C03573=1020.006,186.866,-121.307,168.110,50.738,159.496
C03574=1020.013,187.146,-121.332,168.114,50.729,159.495
C03575=1020.018,187.428,-121.358,168.119,50.721,159.494
C03576=1020.024,187.709,-121.384,168.124,50.713,159.494
C03577=1020.030,187.990,-121.410,168.128,50.705,159.493
C03578=1020.035,188.240,-121.432,168.133,50.698,159.492
C03579=1020.040,188.488,-121.455,168.137,50.691,159.491
C03580=1020.045,188.738,-121.477,168.140,50.683,159.490
C03581=1020.050,188.986,-121.500,168.144,50.676,159.490
C03582=1020.056,189.235,-121.523,168.149,50.669,159.489
C03583=1020.061,189.484,-121.546,168.153,50.662,159.488
C03584=1020.066,189.733,-121.568,168.157,50.654,159.487
C03585=1020.071,189.982,-121.591,168.161,50.647,159.486
C03586=1020.076,190.230,-121.614,168.165,50.640,159.486
C03587=1020.081,190.480,-121.637,168.170,50.633,159.485
C03588=1020.087,190.729,-121.660,168.174,50.626,159.484
C03589=1020.092,190.977,-121.682,168.177,50.619,159.483
C03590=1020.097,191.226,-121.706,168.181,50.611,159.483
C03591=1020.102,191.475,-121.728,168.186,50.604,159.482
C03592=1020.108,191.724,-121.750,168.190,50.597,159.481
C03593=1020.113,191.973,-121.774,168.195,50.590,159.481
C03594=1020.118,192.222,-121.797,168.198,50.583,159.479
C03595=1020.123,192.470,-121.820,168.202,50.576,159.479
C03596=1020.128,192.720,-121.842,168.207,50.569,159.478
C03597=1020.134,192.969,-121.865,168.211,50.561,159.477
C03598=1020.139,193.217,-121.888,168.215,50.554,159.476
C03599=1020.144,193.466,-121.911,168.220,50.547,159.476
C03600=1020.150,193.715,-121.934,168.223,50.540,159.475
C03601=1020.155,193.964,-121.957,168.228,50.533,159.474
C03602=1020.160,194.213,-121.980,168.232,50.526,159.474
C03603=1020.165,194.462,-122.003,168.236,50.518,159.473
C03604=1020.171,194.711,-122.026,168.240,50.511,159.472
C03605=1020.175,194.959,-122.049,168.245,50.504,159.471
C03606=1020.181,195.208,-122.072,168.249,50.497,159.471
C03607=1020.187,195.457,-122.095,168.254,50.490,159.470
C03608=1020.192,195.706,-122.118,168.257,50.483,159.469
C03609=1020.198,195.955,-122.141,168.261,50.475,159.468
C03610=1020.203,196.203,-122.164,168.266,50.468,159.467
C03611=1020.208,196.453,-122.187,168.270,50.461,159.467
C03612=1020.213,196.702,-122.210,168.275,50.454,159.466
C03613=1020.219,196.950,-122.233,168.279,50.447,159.465
C03614=1020.224,197.200,-122.257,168.283,50.439,159.464
C03615=1020.229,197.448,-122.279,168.288,50.432,159.464
C03616=1020.235,197.697,-122.302,168.292,50.425,159.463
C03617=1020.240,197.946,-122.326,168.297,50.418,159.462
C03618=1020.246,198.195,-122.349,168.301,50.411,159.462
C03619=1020.251,198.444,-122.372,168.305,50.403,159.461
C03620=1020.256,198.693,-122.395,168.309,50.396,159.460
C03621=1020.262,198.941,-122.418,168.313,50.389,159.459
C03622=1020.267,199.190,-122.441,168.318,50.382,159.459
C03623=1020.272,199.439,-122.464,168.322,50.375,159.458
C03624=1020.277,199.688,-122.488,168.326,50.368,159.457
C03625=1020.283,199.937,-122.512,168.331,50.361,159.456
C03626=1020.288,200.186,-122.535,168.335,50.354,159.456
C03627=1020.293,200.435,-122.559,168.340,50.347,159.455
C03628=1020.299,200.684,-122.582,168.344,50.340,159.454
C03629=1020.304,200.932,-122.605,168.349,50.333,159.454
C03630=1020.309,201.181,-122.629,168.353,50.326,159.453
C03631=1020.314,201.430,-122.653,168.357,50.319,159.452
C03632=1020.320,201.679,-122.676,168.361,50.312,159.451
C03633=1020.325,201.928,-122.700,168.366,50.305,159.451
C03634=1020.330,202.176,-122.724,168.370,50.298,159.450
C03635=1020.336,202.425,-122.747,168.375,50.291,159.449
C03636=1020.341,202.674,-122.770,168.379,50.284,159.449
C03637=1020.346,202.923,-122.795,168.384,50.277,159.448
C03638=1020.368,203.963,-122.893,168.833,50.371,159.543
C03639=1020.373,204.181,-122.915,168.836,50.366,159.543
C03640=1020.379,204.400,-122.937,168.838,50.360,159.542
C03641=1020.384,204.618,-122.960,168.842,50.355,159.542
C03642=1020.390,204.838,-122.982,168.844,50.349,159.541
C03643=1020.396,205.057,-123.004,168.848,50.344,159.540
C03644=1020.401,205.276,-123.026,168.852,50.339,159.540
C03645=1020.406,205.494,-123.049,168.855,50.333,159.539
C03646=1020.412,205.713,-123.070,168.858,50.328,159.539
C03647=1020.418,205.961,-123.096,168.861,50.322,159.538
C03648=1020.424,206.210,-123.121,168.864,50.316,159.537
C03649=1020.431,206.459,-123.146,168.868,50.310,159.536
C03650=1020.437,206.707,-123.172,168.872,50.304,159.536
C03651=1020.443,206.956,-123.197,168.876,50.298,159.535
C03652=1020.449,207.204,-123.222,168.879,50.292,159.535
C03653=1020.455,207.453,-123.247,168.882,50.287,159.534
C03654=1020.461,207.701,-123.273,168.886,50.281,159.533
C03655=1020.466,207.950,-123.299,168.890,50.275,159.532
C03656=1020.473,208.198,-123.325,168.894,50.269,159.532
C03657=1020.479,208.447,-123.350,168.897,50.263,159.531
C03658=1020.485,208.696,-123.375,168.900,50.257,159.530
C03659=1020.492,208.944,-123.401,168.904,50.251,159.530
C03660=1020.498,209.193,-123.426,168.908,50.245,159.529
C03661=1020.504,209.442,-123.451,168.912,50.239,159.528
C03662=1020.510,209.690,-123.477,168.914,50.233,159.528
C03663=1020.516,209.939,-123.503,168.919,50.228,159.527
C03664=1020.522,210.187,-123.529,168.922,50.222,159.527
C03665=1020.528,210.436,-123.554,168.926,50.216,159.526
C03666=1020.535,210.685,-123.579,168.929,50.210,159.525
C03667=1020.540,210.933,-123.606,168.933,50.205,159.525
C03668=1020.547,211.182,-123.631,168.937,50.199,159.524
C03669=1020.553,211.431,-123.657,168.941,50.193,159.524
C03670=1020.559,211.680,-123.683,168.944,50.187,159.523
C03671=1020.565,211.928,-123.709,168.948,50.182,159.522
C03672=1020.572,212.177,-123.734,168.952,50.176,159.522
C03673=1020.577,212.426,-123.760,168.954,50.170,159.521
C03674=1020.584,212.674,-123.786,168.958,50.164,159.520
C03675=1020.590,212.923,-123.812,168.962,50.159,159.520
C03676=1020.596,213.171,-123.837,168.966,50.153,159.519
C03677=1020.602,213.420,-123.864,168.969,50.147,159.518
C03678=1020.608,213.668,-123.889,168.973,50.142,159.518
C03679=1020.614,213.916,-123.915,168.977,50.136,159.517
C03680=1020.620,214.165,-123.941,168.980,50.130,159.517
C03681=1020.626,214.414,-123.966,168.984,50.125,159.516
C03682=1020.633,214.663,-123.993,168.988,50.119,159.515
C03683=1020.639,214.912,-124.019,168.992,50.114,159.515
C03684=1020.645,215.160,-124.045,168.995,50.108,159.514
C03685=1020.651,215.408,-124.070,168.999,50.102,159.514
C03686=1020.657,215.657,-124.097,169.003,50.097,159.513
C03687=1020.663,215.905,-124.122,169.006,50.091,159.512
C03688=1020.670,216.154,-124.147,169.010,50.086,159.512
C03689=1020.676,216.403,-124.174,169.014,50.080,159.511
C03690=1020.682,216.652,-124.200,169.017,50.074,159.511
C03691=1020.689,216.900,-124.226,169.021,50.069,159.510
C03692=1020.694,217.149,-124.252,169.025,50.063,159.509
C03693=1020.701,217.397,-124.278,169.029,50.058,159.509
C03694=1020.707,217.646,-124.303,169.032,50.052,159.508
C03695=1020.714,217.894,-124.330,169.036,50.047,159.508
C03696=1020.720,218.143,-124.356,169.040,50.041,159.507
C03697=1020.726,218.391,-124.382,169.044,50.035,159.507
C03698=1020.732,218.640,-124.408,169.047,50.030,159.506
C03699=1020.737,218.861,-124.431,169.050,50.025,159.506
C03700=1020.743,219.082,-124.455,169.053,50.020,159.505
C03701=1020.748,219.304,-124.478,169.057,50.015,159.505
C03702=1020.754,219.525,-124.502,169.060,50.011,159.504
C03703=1020.759,219.747,-124.525,169.063,50.006,159.504
C03704=1020.764,219.968,-124.549,169.066,50.001,159.503
C03705=1020.770,220.190,-124.571,169.070,49.996,159.503
C03706=1020.775,220.410,-124.595,169.073,49.991,159.502
C03707=1020.781,220.659,-124.622,169.077,49.986,159.502
C03708=1020.788,220.908,-124.647,169.081,49.981,159.501
C03709=1020.794,221.157,-124.674,169.084,49.976,159.501
C03710=1020.800,221.405,-124.701,169.088,49.970,159.500
C03711=1020.806,221.653,-124.727,169.092,49.965,159.499
C03712=1020.812,221.902,-124.754,169.096,49.960,159.499
C03713=1020.819,222.151,-124.779,169.100,49.954,159.498
C03714=1020.824,222.399,-124.806,169.103,49.949,159.498
C03715=1020.830,222.647,-124.832,169.107,49.943,159.497
C03716=1020.837,222.896,-124.859,169.111,49.938,159.497
C03717=1020.843,223.144,-124.885,169.114,49.933,159.496
C03718=1020.849,223.393,-124.912,169.118,49.927,159.496
C03719=1020.856,223.642,-124.938,169.121,49.922,159.495
C03720=1020.861,223.891,-124.964,169.126,49.917,159.495
C03721=1020.868,224.139,-124.991,169.130,49.912,159.494
C03722=1020.874,224.387,-125.017,169.133,49.907,159.494
C03723=1020.880,224.636,-125.044,169.137,49.901,159.493
C03724=1020.887,224.884,-125.070,169.141,49.895,159.492
C03725=1020.892,225.132,-125.097,169.144,49.890,159.492
C03726=1020.899,225.382,-125.124,169.149,49.885,159.491
C03727=1020.905,225.630,-125.150,169.152,49.880,159.491
C03728=1020.912,225.879,-125.177,169.156,49.875,159.490
C03729=1020.918,226.127,-125.203,169.160,49.870,159.490
C03730=1020.924,226.375,-125.230,169.163,49.865,159.489
C03731=1020.930,226.624,-125.257,169.167,49.859,159.489
C03732=1020.937,226.872,-125.283,169.171,49.853,159.488
C03733=1020.943,227.120,-125.309,169.175,49.849,159.488
C03734=1020.949,227.370,-125.336,169.179,49.844,159.488
C03735=1020.955,227.618,-125.363,169.182,49.839,159.487
C03736=1020.961,227.866,-125.390,169.187,49.834,159.487
C03737=1020.967,228.115,-125.417,169.190,49.829,159.486
C03738=1020.973,228.364,-125.443,169.194,49.824,159.486
C03739=1020.980,228.612,-125.470,169.197,49.819,159.485
C03740=1020.986,228.860,-125.497,169.202,49.813,159.485
C03741=1020.992,229.109,-125.524,169.206,49.808,159.484
C03742=1020.998,229.358,-125.551,169.209,49.803,159.483
C03743=1021.004,229.606,-125.577,169.213,49.798,159.483
C03744=1021.010,229.855,-125.604,169.216,49.793,159.482
C03745=1021.016,230.103,-125.632,169.221,49.788,159.482
C03746=1021.022,230.351,-125.658,169.224,49.783,159.482
C03747=1021.028,230.600,-125.685,169.228,49.778,159.481
C03748=1021.034,230.848,-125.713,169.232,49.773,159.481
C03749=1021.041,231.097,-125.740,169.236,49.768,159.480
C03750=1021.047,231.345,-125.767,169.241,49.763,159.480
C03751=1021.053,231.594,-125.794,169.244,49.758,159.479
C03752=1021.059,231.842,-125.821,169.248,49.753,159.479
C03753=1021.065,232.091,-125.848,169.251,49.748,159.478
C03754=1021.072,232.339,-125.875,169.256,49.744,159.478
C03755=1021.077,232.587,-125.902,169.259,49.739,159.478
C03756=1021.084,232.836,-125.929,169.263,49.733,159.477
C03757=1021.090,233.084,-125.956,169.266,49.728,159.477
C03758=1021.096,233.333,-125.983,169.271,49.724,159.476
C03759=1021.101,233.550,-126.007,169.275,49.720,159.476
C03760=1021.107,233.767,-126.031,169.277,49.716,159.476
C03761=1021.113,233.985,-126.055,169.280,49.711,159.475
C03762=1021.117,234.202,-126.078,169.284,49.706,159.475
C03763=1021.123,234.419,-126.103,169.288,49.702,159.474
C03764=1021.129,234.637,-126.126,169.291,49.698,159.474
C03765=1021.134,234.854,-126.149,169.295,49.694,159.474
C03766=1021.140,235.071,-126.174,169.297,49.690,159.473
C03767=1021.145,235.320,-126.200,169.302,49.684,159.473
C03768=1021.152,235.568,-126.228,169.306,49.680,159.472
C03769=1021.158,235.817,-126.255,169.309,49.675,159.472
C03770=1021.164,236.065,-126.283,169.314,49.670,159.472
C03771=1021.171,236.314,-126.310,169.317,49.665,159.471
C03772=1021.177,236.562,-126.337,169.322,49.661,159.471
C03773=1021.183,236.811,-126.364,169.325,49.656,159.470
C03774=1021.189,237.059,-126.391,169.329,49.651,159.470
C03775=1021.195,237.307,-126.420,169.333,49.646,159.469
C03776=1021.202,237.556,-126.447,169.337,49.641,159.469
C03777=1021.208,237.804,-126.474,169.341,49.637,159.469
C03778=1021.214,238.053,-126.501,169.345,49.632,159.468
C03779=1021.220,238.301,-126.528,169.349,49.627,159.468
C03780=1021.227,238.549,-126.556,169.353,49.622,159.467
C03781=1021.233,238.798,-126.583,169.356,49.618,159.467
C03782=1021.239,239.046,-126.611,169.361,49.613,159.466
C03783=1021.246,239.295,-126.638,169.364,49.609,159.466
C03784=1021.251,239.543,-126.666,169.369,49.604,159.466
C03785=1021.258,239.792,-126.693,169.372,49.599,159.465
C03786=1021.264,240.040,-126.722,169.377,49.594,159.465
C03787=1021.270,240.288,-126.749,169.380,49.590,159.465
C03788=1021.276,240.537,-126.777,169.385,49.585,159.464
C03789=1021.282,240.785,-126.805,169.388,49.581,159.464
C03790=1021.289,241.033,-126.832,169.393,49.576,159.464
C03791=1021.295,241.282,-126.859,169.396,49.571,159.463
C03792=1021.301,241.531,-126.888,169.400,49.567,159.463
C03793=1021.307,241.779,-126.915,169.404,49.562,159.462
C03794=1021.313,242.027,-126.943,169.408,49.558,159.462
C03795=1021.320,242.276,-126.971,169.412,49.553,159.462
C03796=1021.326,242.524,-126.998,169.416,49.549,159.461
C03797=1021.332,242.772,-127.027,169.420,49.544,159.461
C03798=1021.338,243.021,-127.055,169.424,49.540,159.461
C03799=1021.344,243.268,-127.082,169.429,49.535,159.460
C03800=1021.350,243.517,-127.110,169.432,49.530,159.460
C03801=1021.357,243.766,-127.138,169.436,49.526,159.460
C03802=1021.362,244.014,-127.166,169.440,49.522,159.459
C03803=1021.368,244.262,-127.194,169.444,49.517,159.459
C03804=1021.375,244.511,-127.222,169.448,49.513,159.459
C03805=1021.381,244.760,-127.250,169.452,49.509,159.458
C03806=1021.386,245.008,-127.278,169.456,49.504,159.458
C03807=1021.393,245.256,-127.307,169.460,49.500,159.458
C03808=1021.399,245.504,-127.335,169.464,49.496,159.457
C03809=1021.404,245.752,-127.363,169.468,49.491,159.457
C03810=1021.411,246.001,-127.391,169.472,49.487,159.457
C03811=1021.417,246.250,-127.419,169.477,49.482,159.456
C03812=1021.423,246.498,-127.448,169.480,49.478,159.456
C03813=1021.429,246.745,-127.475,169.485,49.473,159.456
C03814=1021.435,246.994,-127.504,169.488,49.469,159.455
C03815=1021.441,247.243,-127.532,169.492,49.465,159.455
C03816=1021.448,247.491,-127.561,169.497,49.460,159.455
C03817=1021.454,247.740,-127.589,169.500,49.456,159.454
C03818=1021.460,247.988,-127.617,169.505,49.452,159.454
C03819=1021.465,248.202,-127.641,169.508,49.448,159.454
C03820=1021.470,248.416,-127.665,169.511,49.444,159.453
C03821=1021.476,248.630,-127.690,169.515,49.441,159.453
C03822=1021.482,248.844,-127.714,169.518,49.437,159.453
C03823=1021.486,249.058,-127.739,169.522,49.433,159.453
C03824=1021.492,249.273,-127.763,169.526,49.430,159.452
C03825=1021.497,249.487,-127.787,169.529,49.426,159.452
C03826=1021.503,249.701,-127.812,169.532,49.422,159.452
C03827=1021.509,249.950,-127.840,169.536,49.419,159.452
C03828=1021.515,250.197,-127.869,169.541,49.414,159.451
C03829=1021.521,250.445,-127.897,169.545,49.410,159.451
C03830=1021.527,250.694,-127.925,169.549,49.405,159.451
C03831=1021.533,250.942,-127.954,169.553,49.401,159.450
C03832=1021.540,251.191,-127.982,169.558,49.396,159.450
C03833=1021.546,251.439,-128.011,169.562,49.393,159.450
C03834=1021.552,251.688,-128.039,169.565,49.389,159.450
C03835=1021.559,251.936,-128.067,169.570,49.384,159.449
C03836=1021.565,252.184,-128.096,169.573,49.380,159.449
C03837=1021.571,252.433,-128.124,169.578,49.375,159.449
C03838=1021.578,252.680,-128.152,169.582,49.372,159.449
C03839=1021.584,252.929,-128.181,169.587,49.367,159.448
C03840=1021.590,253.177,-128.210,169.590,49.363,159.448
C03841=1021.596,253.425,-128.237,169.594,49.359,159.448
C03842=1021.603,253.674,-128.267,169.599,49.355,159.447
C03843=1021.609,253.922,-128.295,169.602,49.351,159.447
C03844=1021.616,254.170,-128.323,169.607,49.346,159.447
C03845=1021.622,254.418,-128.352,169.611,49.343,159.447
C03846=1021.628,254.667,-128.381,169.616,49.338,159.446
C03847=1021.634,254.915,-128.410,169.619,49.334,159.446
C03848=1021.641,255.164,-128.437,169.624,49.329,159.446
C03849=1021.647,255.412,-128.466,169.628,49.326,159.446
C03850=1021.653,255.660,-128.496,169.631,49.322,159.445
C03851=1021.660,255.908,-128.523,169.636,49.318,159.445
C03852=1021.666,256.156,-128.552,169.640,49.314,159.445
C03853=1021.672,256.405,-128.581,169.645,49.309,159.444
C03854=1021.679,256.653,-128.609,169.649,49.306,159.444
C03855=1021.685,256.901,-128.638,169.653,49.301,159.444
C03856=1021.692,257.151,-128.667,169.657,49.297,159.444
C03857=1021.699,257.398,-128.695,169.662,49.293,159.444
C03858=1021.705,257.647,-128.724,169.666,49.289,159.443
C03859=1021.711,257.895,-128.753,169.670,49.285,159.443
C03860=1021.717,258.143,-128.782,169.674,49.281,159.443
C03861=1021.724,258.391,-128.810,169.678,49.277,159.443
C03862=1021.731,258.639,-128.839,169.683,49.273,159.442
C03863=1021.737,258.887,-128.868,169.687,49.269,159.442
C03864=1021.744,259.136,-128.896,169.691,49.265,159.442
C03865=1021.750,259.384,-128.925,169.695,49.260,159.442
C03866=1021.757,259.633,-128.954,169.700,49.256,159.441
C03867=1021.764,259.881,-128.983,169.704,49.252,159.441
C03868=1021.770,260.129,-129.012,169.709,49.248,159.441
C03869=1021.776,260.377,-129.041,169.713,49.245,159.441
C03870=1021.782,260.625,-129.070,169.716,49.241,159.440
C03871=1021.789,260.873,-129.099,169.721,49.237,159.440
C03872=1021.795,261.121,-129.128,169.725,49.233,159.440
C03873=1021.801,261.369,-129.157,169.730,49.229,159.440
C03874=1021.807,261.618,-129.186,169.734,49.225,159.440
C03875=1021.813,261.867,-129.216,169.738,49.222,159.440
C03876=1021.820,262.115,-129.245,169.743,49.218,159.439
C03877=1021.826,262.363,-129.274,169.746,49.214,159.439
C03878=1021.832,262.611,-129.303,169.750,49.210,159.439
C03879=1021.838,262.824,-129.328,169.754,49.207,159.439
C03880=1021.843,263.038,-129.354,169.759,49.204,159.439
C03881=1021.849,263.251,-129.379,169.762,49.200,159.439
C03882=1021.854,263.464,-129.404,169.766,49.197,159.438
C03883=1021.860,263.678,-129.429,169.770,49.193,159.438
C03884=1021.865,263.891,-129.454,169.773,49.191,159.438
C03885=1021.870,264.104,-129.479,169.777,49.187,159.438
C03886=1021.876,264.318,-129.505,169.781,49.184,159.438
C03887=1021.882,264.566,-129.534,169.785,49.180,159.438
C03888=1021.888,264.814,-129.563,169.789,49.177,159.437
C03889=1021.895,265.062,-129.593,169.794,49.173,159.437
C03890=1021.901,265.310,-129.622,169.798,49.169,159.437
C03891=1021.908,265.559,-129.652,169.803,49.165,159.437
C03892=1021.914,265.807,-129.681,169.807,49.162,159.437
C03893=1021.920,266.055,-129.711,169.810,49.158,159.437
C03894=1021.926,266.303,-129.740,169.815,49.154,159.436
C03895=1021.933,266.552,-129.769,169.819,49.150,159.436
C03896=1021.940,266.799,-129.799,169.823,49.147,159.436
C03897=1021.945,267.048,-129.829,169.828,49.143,159.436
C03898=1021.952,267.296,-129.859,169.832,49.139,159.436
C03899=1021.958,267.544,-129.888,169.837,49.136,159.436
C03900=1021.965,267.792,-129.917,169.841,49.132,159.436
C03901=1021.971,268.040,-129.947,169.846,49.129,159.436
C03902=1021.977,268.289,-129.977,169.851,49.125,159.435
C03903=1021.984,268.536,-130.007,169.855,49.122,159.435
C03904=1021.989,268.785,-130.036,169.860,49.118,159.435
C03905=1021.997,269.033,-130.066,169.864,49.114,159.435
C03906=1022.003,269.281,-130.095,169.868,49.111,159.435
C03907=1022.009,269.528,-130.125,169.873,49.107,159.435
C03908=1022.016,269.778,-130.155,169.877,49.104,159.435
C03909=1022.022,270.025,-130.185,169.882,49.100,159.434
C03910=1022.028,270.273,-130.215,169.886,49.097,159.435
C03911=1022.035,270.522,-130.245,169.890,49.093,159.434
C03912=1022.041,270.770,-130.275,169.895,49.089,159.434
C03913=1022.047,271.017,-130.305,169.899,49.086,159.434
C03914=1022.054,271.266,-130.334,169.903,49.082,159.434
C03915=1022.060,271.514,-130.365,169.908,49.079,159.434
C03916=1022.067,271.762,-130.395,169.912,49.076,159.434
C03917=1022.072,272.010,-130.424,169.917,49.072,159.434
C03918=1022.079,272.258,-130.454,169.921,49.068,159.434
C03919=1022.085,272.506,-130.485,169.926,49.066,159.434
C03920=1022.092,272.754,-130.514,169.931,49.062,159.433
C03921=1022.098,273.003,-130.544,169.935,49.058,159.433
C03922=1022.105,273.251,-130.574,169.939,49.055,159.433
C03923=1022.110,273.498,-130.605,169.944,49.051,159.433
C03924=1022.118,273.747,-130.635,169.948,49.048,159.433
C03925=1022.123,273.995,-130.665,169.953,49.045,159.433
C03926=1022.131,274.243,-130.695,169.957,49.041,159.433
C03927=1022.136,274.491,-130.725,169.961,49.038,159.433
C03928=1022.143,274.739,-130.755,169.967,49.035,159.433
C03929=1022.149,274.987,-130.785,169.971,49.031,159.433
C03930=1022.156,275.236,-130.816,169.975,49.028,159.433
C03931=1022.162,275.483,-130.846,169.980,49.024,159.433
C03932=1022.169,275.732,-130.876,169.984,49.021,159.433
C03933=1022.175,275.979,-130.906,169.989,49.018,159.433
C03934=1022.181,276.228,-130.937,169.993,49.014,159.432
C03935=1022.188,276.475,-130.967,169.998,49.011,159.432
C03936=1022.194,276.724,-130.997,170.003,49.007,159.432
C03937=1022.201,276.971,-131.027,170.007,49.005,159.432
C03938=1022.207,277.220,-131.058,170.012,49.001,159.432
C03939=1022.213,277.435,-131.085,170.015,48.998,159.432
C03940=1022.218,277.651,-131.111,170.020,48.995,159.432
C03941=1022.223,277.867,-131.138,170.024,48.993,159.432
C03942=1022.230,278.082,-131.164,170.027,48.990,159.432
C03943=1022.235,278.298,-131.191,170.032,48.987,159.432
C03944=1022.240,278.514,-131.217,170.036,48.984,159.432
C03945=1022.245,278.729,-131.244,170.039,48.982,159.432
C03946=1022.251,278.945,-131.271,170.044,48.979,159.432
C03947=1022.258,279.192,-131.301,170.048,48.976,159.432
C03948=1022.264,279.440,-131.332,170.053,48.972,159.432
C03949=1022.271,279.689,-131.362,170.057,48.969,159.432
C03950=1022.277,279.937,-131.393,170.062,48.966,159.432
C03951=1022.283,280.185,-131.424,170.067,48.963,159.432
C03952=1022.290,280.432,-131.454,170.071,48.960,159.432
C03953=1022.296,280.681,-131.485,170.076,48.957,159.432
C03954=1022.303,280.929,-131.515,170.081,48.954,159.432
C03955=1022.309,281.176,-131.547,170.085,48.951,159.432
C03956=1022.315,281.425,-131.577,170.090,48.947,159.432
C03957=1022.322,281.673,-131.607,170.094,48.944,159.432
C03958=1022.328,281.920,-131.638,170.099,48.941,159.432
C03959=1022.335,282.169,-131.669,170.104,48.938,159.432
C03960=1022.342,282.417,-131.701,170.108,48.935,159.432
C03961=1022.347,282.665,-131.731,170.113,48.932,159.432
C03962=1022.355,282.913,-131.761,170.118,48.929,159.432
C03963=1022.361,283.161,-131.792,170.122,48.926,159.432
C03964=1022.368,283.409,-131.823,170.127,48.923,159.432
C03965=1022.374,283.656,-131.854,170.132,48.920,159.432
C03966=1022.380,283.905,-131.885,170.137,48.917,159.432
C03967=1022.387,284.153,-131.916,170.141,48.913,159.432
C03968=1022.394,284.400,-131.946,170.146,48.910,159.432
C03969=1022.400,284.648,-131.978,170.151,48.907,159.432
C03970=1022.407,284.897,-132.008,170.155,48.904,159.432
C03971=1022.413,285.145,-132.040,170.161,48.901,159.432
C03972=1022.420,285.393,-132.071,170.165,48.898,159.432
C03973=1022.426,285.640,-132.102,170.170,48.895,159.432
C03974=1022.433,285.888,-132.133,170.175,48.892,159.432
C03975=1022.439,286.136,-132.164,170.179,48.889,159.432
C03976=1022.446,286.385,-132.195,170.184,48.886,159.432
C03977=1022.452,286.632,-132.226,170.189,48.883,159.432
C03978=1022.459,286.880,-132.258,170.194,48.880,159.432
C03979=1022.465,287.128,-132.288,170.199,48.878,159.433
C03980=1022.472,287.376,-132.320,170.203,48.875,159.433
C03981=1022.479,287.624,-132.351,170.208,48.872,159.433
C03982=1022.485,287.871,-132.382,170.213,48.869,159.433
C03983=1022.491,288.119,-132.414,170.218,48.866,159.433
C03984=1022.498,288.368,-132.444,170.222,48.863,159.433
C03985=1022.505,288.616,-132.476,170.227,48.860,159.433
C03986=1022.511,288.864,-132.508,170.232,48.858,159.433
C03987=1022.517,289.112,-132.539,170.237,48.855,159.433
C03988=1022.524,289.360,-132.571,170.242,48.852,159.433
C03989=1022.530,289.607,-132.602,170.246,48.849,159.433
C03990=1022.537,289.855,-132.633,170.251,48.846,159.433
C03991=1022.544,290.103,-132.665,170.257,48.844,159.433
C03992=1022.550,290.351,-132.696,170.261,48.841,159.433
C03993=1022.557,290.599,-132.728,170.266,48.838,159.434
C03994=1022.563,290.847,-132.760,170.271,48.835,159.434
C03995=1022.570,291.095,-132.791,170.276,48.832,159.434
C03996=1022.576,291.343,-132.822,170.281,48.829,159.434
C03997=1022.583,291.591,-132.854,170.285,48.827,159.434
C03998=1022.590,291.838,-132.885,170.291,48.824,159.434
C03999=1022.595,292.060,-132.914,170.295,48.821,159.434
C04000=1022.601,292.281,-132.942,170.299,48.819,159.434
C04001=1022.607,292.504,-132.971,170.303,48.817,159.434
C04002=1022.614,292.725,-132.999,170.308,48.814,159.434
C04003=1022.619,292.947,-133.027,170.312,48.812,159.435
C04004=1022.625,293.168,-133.055,170.317,48.809,159.435
C04005=1022.631,293.390,-133.084,170.321,48.807,159.435
C04006=1022.637,293.613,-133.112,170.326,48.805,159.435
C04007=1022.643,293.860,-133.144,170.330,48.802,159.435
C04008=1022.649,294.109,-133.176,170.335,48.800,159.435
C04009=1022.656,294.356,-133.208,170.341,48.797,159.435
C04010=1022.662,294.604,-133.240,170.345,48.795,159.435
C04011=1022.669,294.852,-133.272,170.350,48.792,159.436
C04012=1022.675,295.100,-133.305,170.355,48.789,159.436
C04013=1022.681,295.348,-133.337,170.360,48.787,159.436
C04014=1022.688,295.595,-133.369,170.366,48.785,159.436
C04015=1022.694,295.843,-133.401,170.370,48.782,159.436
C04016=1022.701,296.090,-133.433,170.375,48.780,159.436
C04017=1022.707,296.339,-133.465,170.380,48.777,159.437
C04018=1022.714,296.586,-133.498,170.385,48.774,159.437
C04019=1022.720,296.834,-133.529,170.390,48.772,159.437
C04020=1022.727,297.082,-133.562,170.395,48.769,159.437
C04021=1022.733,297.330,-133.593,170.400,48.767,159.437
C04022=1022.740,297.577,-133.626,170.405,48.764,159.437
C04023=1022.746,297.825,-133.659,170.410,48.762,159.438
C04024=1022.753,298.073,-133.690,170.416,48.759,159.438
C04025=1022.759,298.320,-133.723,170.420,48.757,159.438
C04026=1022.766,298.569,-133.755,170.425,48.754,159.438
C04027=1022.773,298.817,-133.788,170.430,48.752,159.438
C04028=1022.779,299.064,-133.820,170.435,48.750,159.439
C04029=1022.786,299.312,-133.852,170.441,48.747,159.439
C04030=1022.792,299.560,-133.884,170.445,48.745,159.439
C04031=1022.799,299.807,-133.917,170.451,48.743,159.439
C04032=1022.805,300.055,-133.949,170.456,48.740,159.440
C04033=1022.812,300.303,-133.982,170.461,48.737,159.440
C04034=1022.819,300.551,-134.014,170.466,48.735,159.440
C04035=1022.825,300.798,-134.047,170.470,48.733,159.440
C04036=1022.832,301.046,-134.079,170.476,48.730,159.440
C04037=1022.839,301.295,-134.111,170.481,48.728,159.440
C04038=1022.845,301.542,-134.144,170.487,48.726,159.441
C04039=1022.852,301.789,-134.176,170.491,48.724,159.441
C04040=1022.858,302.037,-134.209,170.497,48.721,159.441
C04041=1022.865,302.285,-134.242,170.502,48.719,159.441
C04042=1022.872,302.533,-134.274,170.507,48.716,159.442
C04043=1022.879,302.780,-134.307,170.512,48.714,159.442
C04044=1022.886,303.027,-134.339,170.518,48.712,159.442
C04045=1022.892,303.276,-134.371,170.522,48.709,159.442
C04046=1022.898,303.524,-134.404,170.528,48.707,159.443
C04047=1022.905,303.771,-134.436,170.533,48.705,159.443
C04048=1022.912,304.020,-134.469,170.539,48.702,159.443
C04049=1022.919,304.267,-134.502,170.543,48.700,159.443
C04050=1022.926,304.514,-134.534,170.549,48.698,159.443
C04051=1022.933,304.763,-134.567,170.554,48.695,159.444
C04052=1022.940,305.010,-134.600,170.559,48.693,159.444
C04053=1022.947,305.258,-134.633,170.564,48.691,159.444
C04054=1022.953,305.505,-134.666,170.570,48.689,159.445
C04055=1022.960,305.753,-134.698,170.575,48.687,159.445
C04056=1022.967,306.001,-134.731,170.580,48.684,159.445
C04057=1022.973,306.248,-134.764,170.585,48.682,159.445
C04058=1022.981,306.496,-134.797,170.591,48.680,159.445
C04059=1022.987,306.727,-134.827,170.596,48.678,159.446
C04060=1022.993,306.958,-134.858,170.601,48.676,159.446
C04061=1023.000,307.188,-134.889,170.605,48.674,159.446
C04062=1023.006,307.418,-134.919,170.610,48.671,159.446
C04063=1023.013,307.648,-134.949,170.615,48.670,159.447
C04064=1023.019,307.879,-134.979,170.621,48.667,159.447
C04065=1023.025,308.109,-135.011,170.625,48.665,159.447
C04066=1023.032,308.340,-135.041,170.630,48.664,159.448
C04067=1023.039,308.588,-135.074,170.636,48.661,159.448
C04068=1023.046,308.835,-135.106,170.641,48.659,159.448
C04069=1023.053,309.083,-135.140,170.647,48.657,159.449
C04070=1023.060,309.330,-135.172,170.651,48.655,159.449
C04071=1023.067,309.578,-135.206,170.657,48.652,159.449
C04072=1023.073,309.825,-135.239,170.662,48.651,159.449
C04073=1023.081,310.073,-135.272,170.668,48.648,159.450
C04074=1023.088,310.321,-135.305,170.674,48.646,159.450
C04075=1023.094,310.569,-135.338,170.679,48.644,159.450
C04076=1023.102,310.816,-135.372,170.684,48.643,159.451
C04077=1023.108,311.064,-135.406,170.689,48.640,159.451
C04078=1023.114,311.312,-135.439,170.694,48.639,159.451
C04079=1023.121,311.559,-135.473,170.700,48.637,159.452
C04080=1023.128,311.807,-135.506,170.705,48.635,159.452
C04081=1023.134,312.054,-135.540,170.711,48.633,159.452
C04082=1023.141,312.302,-135.574,170.716,48.631,159.453
C04083=1023.148,312.549,-135.607,170.722,48.629,159.453
C04084=1023.154,312.797,-135.641,170.727,48.627,159.453
C04085=1023.161,313.045,-135.675,170.733,48.626,159.454
C04086=1023.168,313.292,-135.708,170.738,48.623,159.454
C04087=1023.175,313.540,-135.742,170.744,48.622,159.454
C04088=1023.181,313.787,-135.776,170.750,48.620,159.455
C04089=1023.188,314.035,-135.810,170.755,48.618,159.455
C04090=1023.195,314.283,-135.844,170.761,48.616,159.456
C04091=1023.202,314.530,-135.877,170.766,48.614,159.456
C04092=1023.208,314.778,-135.911,170.772,48.612,159.456
C04093=1023.215,315.025,-135.945,170.777,48.611,159.457
C04094=1023.222,315.272,-135.979,170.783,48.609,159.457
C04095=1023.228,315.520,-136.013,170.788,48.607,159.458
C04096=1023.236,315.768,-136.047,170.794,48.605,159.458
C04097=1023.243,316.016,-136.081,170.798,48.603,159.458
C04098=1023.249,316.263,-136.114,170.804,48.601,159.459
C04099=1023.256,316.511,-136.149,170.810,48.600,159.459
C04100=1023.263,316.758,-136.182,170.815,48.598,159.460
C04101=1023.270,317.006,-136.216,170.822,48.596,159.460
C04102=1023.276,317.253,-136.250,170.827,48.595,159.460
C04103=1023.283,317.501,-136.284,170.833,48.593,159.461
C04104=1023.290,317.749,-136.318,170.838,48.591,159.461
C04105=1023.298,317.996,-136.352,170.844,48.589,159.462
C04106=1023.304,318.244,-136.386,170.850,48.588,159.462
C04107=1023.312,318.491,-136.421,170.855,48.586,159.462
C04108=1023.318,318.738,-136.454,170.861,48.584,159.463
C04109=1023.325,318.986,-136.489,170.866,48.583,159.463
C04110=1023.332,319.234,-136.522,170.872,48.581,159.464
C04111=1023.339,319.482,-136.556,170.878,48.579,159.464
C04112=1023.346,319.729,-136.591,170.883,48.577,159.465
C04113=1023.353,319.977,-136.625,170.889,48.576,159.465
C04114=1023.360,320.224,-136.659,170.895,48.574,159.466
C04115=1023.367,320.472,-136.693,170.900,48.573,159.466
C04116=1023.374,320.719,-136.728,170.906,48.571,159.466
C04117=1023.381,320.967,-136.762,170.911,48.569,159.467
C04118=1023.389,321.215,-136.796,170.917,48.568,159.467
C04119=1023.395,321.447,-136.828,170.922,48.566,159.468
C04120=1023.402,321.680,-136.860,170.929,48.565,159.468
C04121=1023.408,321.914,-136.893,170.934,48.563,159.469
C04122=1023.414,322.146,-136.925,170.939,48.562,159.469
C04123=1023.421,322.379,-136.958,170.945,48.560,159.469
C04124=1023.428,322.613,-136.990,170.950,48.558,159.470
C04125=1023.436,322.846,-137.022,170.955,48.557,159.470
C04126=1023.442,323.078,-137.054,170.961,48.556,159.471
C04127=1023.448,323.326,-137.089,170.966,48.554,159.471
C04128=1023.456,323.574,-137.124,170.973,48.553,159.472
C04129=1023.464,323.821,-137.158,170.979,48.551,159.472
C04130=1023.470,324.069,-137.193,170.985,48.549,159.473
C04131=1023.478,324.316,-137.227,170.990,48.548,159.473
C04132=1023.485,324.563,-137.262,170.996,48.546,159.474
C04133=1023.492,324.811,-137.296,171.002,48.545,159.474
C04134=1023.499,325.058,-137.331,171.008,48.544,159.475
C04135=1023.507,325.307,-137.365,171.014,48.542,159.475
C04136=1023.514,325.554,-137.400,171.020,48.540,159.476
C04137=1023.521,325.801,-137.434,171.026,48.539,159.476
C04138=1023.528,326.049,-137.468,171.031,48.537,159.477
C04139=1023.535,326.296,-137.503,171.038,48.536,159.477
C04140=1023.543,326.544,-137.538,171.044,48.534,159.478
C04141=1023.551,326.791,-137.573,171.049,48.533,159.478
C04142=1023.558,327.038,-137.608,171.055,48.531,159.479
C04143=1023.565,327.286,-137.642,171.061,48.530,159.479
C04144=1023.572,327.533,-137.677,171.068,48.529,159.480
C04145=1023.579,327.781,-137.712,171.073,48.527,159.480
C04146=1023.586,328.028,-137.748,171.079,48.526,159.481
C04147=1023.594,328.275,-137.783,171.086,48.525,159.482
C04148=1023.600,328.522,-137.818,171.091,48.523,159.482
C04149=1023.607,328.770,-137.853,171.097,48.522,159.483
C04150=1023.614,329.018,-137.889,171.103,48.521,159.483
C04151=1023.622,329.265,-137.923,171.110,48.520,159.484
C04152=1023.629,329.512,-137.958,171.115,48.519,159.485
C04153=1023.636,329.760,-137.994,171.121,48.517,159.485
C04154=1023.643,330.008,-138.029,171.127,48.516,159.486
C04155=1023.650,330.254,-138.065,171.133,48.515,159.486
C04156=1023.658,330.502,-138.100,171.139,48.514,159.487
C04157=1023.665,330.750,-138.135,171.146,48.512,159.487
C04158=1023.672,330.997,-138.170,171.152,48.511,159.488
C04159=1023.679,331.245,-138.205,171.158,48.510,159.489
C04160=1023.686,331.492,-138.241,171.163,48.508,159.489
C04161=1023.694,331.739,-138.276,171.170,48.507,159.490
C04162=1023.701,331.987,-138.311,171.176,48.506,159.490
C04163=1023.708,332.234,-138.347,171.182,48.505,159.491
C04164=1023.715,332.482,-138.383,171.188,48.504,159.492
C04165=1023.723,332.729,-138.417,171.194,48.503,159.492
C04166=1023.731,332.976,-138.453,171.201,48.501,159.493
C04167=1023.737,333.224,-138.489,171.207,48.500,159.494
C04168=1023.745,333.471,-138.525,171.213,48.499,159.494
C04169=1023.752,333.718,-138.560,171.219,48.499,159.495
C04170=1023.759,333.965,-138.596,171.225,48.497,159.496
C04171=1023.766,334.213,-138.631,171.232,48.496,159.496
C04172=1023.773,334.460,-138.667,171.238,48.495,159.497
C04173=1023.781,334.707,-138.703,171.244,48.494,159.497
C04174=1023.788,334.955,-138.739,171.250,48.493,159.498
C04175=1023.795,335.202,-138.775,171.257,48.492,159.499
C04176=1023.803,335.450,-138.811,171.263,48.491,159.499
C04177=1023.810,335.697,-138.846,171.269,48.490,159.500
C04178=1023.818,335.944,-138.882,171.276,48.489,159.501
C04179=1023.824,336.175,-138.916,171.281,48.488,159.502
C04180=1023.831,336.406,-138.950,171.287,48.487,159.502
C04181=1023.838,336.637,-138.983,171.293,48.486,159.503
C04182=1023.844,336.867,-139.016,171.299,48.485,159.503
C04183=1023.852,337.098,-139.050,171.305,48.485,159.504
C04184=1023.858,337.329,-139.084,171.311,48.484,159.505
C04185=1023.865,337.560,-139.117,171.317,48.483,159.505
C04186=1023.872,337.790,-139.151,171.322,48.482,159.506
C04187=1023.880,338.037,-139.187,171.329,48.481,159.507
C04188=1023.887,338.285,-139.222,171.336,48.480,159.507
C04189=1023.894,338.533,-139.259,171.342,48.479,159.508
C04190=1023.901,338.780,-139.295,171.349,48.478,159.509
C04191=1023.908,339.027,-139.331,171.354,48.478,159.510
C04192=1023.916,339.274,-139.367,171.361,48.476,159.510
C04193=1023.924,339.522,-139.404,171.367,48.476,159.511
C04194=1023.932,339.769,-139.440,171.374,48.475,159.512
C04195=1023.939,340.016,-139.476,171.380,48.474,159.512
C04196=1023.947,340.263,-139.513,171.387,48.473,159.513
C04197=1023.954,340.510,-139.549,171.394,48.472,159.514
C04198=1023.961,340.758,-139.586,171.400,48.472,159.515
C04199=1023.968,341.005,-139.622,171.407,48.470,159.515
C04200=1023.976,341.252,-139.659,171.413,48.470,159.516
C04201=1023.983,341.499,-139.695,171.419,48.469,159.517
C04202=1023.991,341.747,-139.731,171.425,48.468,159.518
C04203=1023.999,341.994,-139.768,171.432,48.468,159.518
C04204=1024.006,342.241,-139.805,171.439,48.467,159.519
C04205=1024.013,342.488,-139.841,171.446,48.466,159.520
C04206=1024.021,342.735,-139.878,171.452,48.466,159.521
C04207=1024.028,342.983,-139.915,171.459,48.465,159.522
C04208=1024.035,343.230,-139.951,171.465,48.464,159.522
C04209=1024.043,343.477,-139.988,171.472,48.463,159.523
C04210=1024.050,343.725,-140.025,171.479,48.463,159.524
C04211=1024.058,343.971,-140.062,171.486,48.462,159.525
C04212=1024.065,344.219,-140.099,171.492,48.462,159.526
C04213=1024.073,344.466,-140.135,171.499,48.461,159.526
C04214=1024.080,344.713,-140.171,171.506,48.460,159.527
C04215=1024.088,344.960,-140.209,171.512,48.460,159.528
C04216=1024.096,345.207,-140.246,171.519,48.459,159.529
C04217=1024.103,345.454,-140.283,171.526,48.459,159.530
C04218=1024.110,345.701,-140.320,171.533,48.458,159.531
C04219=1024.118,345.948,-140.356,171.539,48.457,159.531
C04220=1024.126,346.197,-140.394,171.546,48.457,159.532
C04221=1024.134,346.443,-140.431,171.553,48.456,159.533
C04222=1024.141,346.690,-140.468,171.559,48.456,159.534
C04223=1024.149,346.937,-140.505,171.566,48.455,159.535
C04224=1024.157,347.185,-140.541,171.573,48.454,159.536
C04225=1024.164,347.432,-140.579,171.579,48.454,159.536
C04226=1024.172,347.679,-140.616,171.587,48.454,159.537
C04227=1024.179,347.926,-140.653,171.593,48.453,159.538
C04228=1024.187,348.173,-140.690,171.600,48.452,159.539
C04229=1024.195,348.420,-140.728,171.607,48.452,159.540
C04230=1024.202,348.667,-140.765,171.614,48.452,159.541
C04231=1024.210,348.914,-140.802,171.620,48.451,159.542
C04232=1024.218,349.162,-140.840,171.627,48.451,159.543
C04233=1024.226,349.408,-140.877,171.634,48.451,159.544
C04234=1024.233,349.656,-140.914,171.641,48.450,159.544
C04235=1024.240,349.903,-140.952,171.648,48.449,159.545
C04236=1024.248,350.149,-140.990,171.655,48.449,159.546
C04237=1024.256,350.397,-141.028,171.661,48.449,159.547
C04238=1024.264,350.644,-141.065,171.668,48.449,159.548
C04239=1024.270,350.873,-141.100,171.675,48.448,159.549
C04240=1024.278,351.102,-141.135,171.682,48.448,159.550
C04241=1024.286,351.332,-141.170,171.688,48.448,159.551
C04242=1024.292,351.561,-141.204,171.695,48.447,159.551
C04243=1024.299,351.790,-141.240,171.701,48.447,159.552
C04244=1024.306,352.019,-141.274,171.708,48.447,159.553
C04245=1024.314,352.249,-141.309,171.714,48.446,159.554
C04246=1024.322,352.477,-141.344,171.721,48.446,159.555
C04247=1024.329,352.724,-141.382,171.728,48.446,159.556
C04248=1024.337,352.972,-141.420,171.735,48.446,159.557
C04249=1024.345,353.218,-141.457,171.742,48.446,159.558
C04250=1024.352,353.465,-141.495,171.750,48.445,159.559
C04251=1024.360,353.713,-141.533,171.757,48.445,159.560
C04252=1024.369,353.959,-141.571,171.764,48.445,159.561
C04253=1024.376,354.207,-141.609,171.770,48.444,159.562
C04254=1024.384,354.453,-141.647,171.778,48.444,159.563
C04255=1024.391,354.701,-141.685,171.785,48.444,159.564
C04256=1024.399,354.948,-141.723,171.793,48.444,159.565
C04257=1024.408,355.194,-141.761,171.800,48.444,159.566
C04258=1024.415,355.442,-141.799,171.807,48.444,159.567
C04259=1024.423,355.688,-141.837,171.813,48.443,159.568
C04260=1024.431,355.936,-141.876,171.820,48.443,159.569
C04261=1024.439,356.182,-141.914,171.829,48.443,159.570
C04262=1024.447,356.430,-141.952,171.836,48.443,159.571
C04263=1024.454,356.676,-141.990,171.843,48.443,159.572
C04264=1024.463,356.923,-142.028,171.850,48.443,159.573
C04265=1024.471,357.170,-142.066,171.858,48.443,159.574
C04266=1024.479,357.417,-142.105,171.865,48.443,159.575
C04267=1024.486,357.664,-142.143,171.872,48.443,159.576
C04268=1024.494,357.911,-142.182,171.879,48.443,159.577
C04269=1024.503,358.158,-142.220,171.887,48.443,159.578
C04270=1024.510,358.404,-142.259,171.894,48.443,159.579
C04271=1024.518,358.652,-142.297,171.901,48.443,159.580
C04272=1024.526,358.899,-142.336,171.909,48.442,159.581
C04273=1024.534,359.145,-142.374,171.916,48.442,159.582
C04274=1024.542,359.393,-142.413,171.924,48.442,159.583
C04275=1024.550,359.640,-142.451,171.931,48.443,159.585
C04276=1024.559,359.885,-142.490,171.939,48.443,159.586
C04277=1024.567,360.133,-142.528,171.946,48.443,159.587
C04278=1024.574,360.380,-142.567,171.953,48.443,159.588
C04279=1024.582,360.627,-142.606,171.961,48.443,159.589
C04280=1024.590,360.873,-142.645,171.969,48.443,159.590
C04281=1024.599,361.121,-142.684,171.976,48.444,159.591
C04282=1024.607,361.367,-142.723,171.984,48.443,159.592
C04283=1024.614,361.614,-142.762,171.991,48.444,159.594
C04284=1024.622,361.861,-142.801,171.998,48.444,159.595
C04285=1024.630,362.108,-142.840,172.007,48.444,159.596
C04286=1024.639,362.354,-142.879,172.014,48.444,159.597
C04287=1024.646,362.601,-142.917,172.022,48.444,159.598
C04288=1024.654,362.848,-142.957,172.030,48.445,159.599
C04289=1024.662,363.095,-142.996,172.037,48.445,159.600
C04290=1024.671,363.342,-143.035,172.045,48.445,159.602
C04291=1024.679,363.588,-143.074,172.052,48.445,159.603
C04292=1024.687,363.835,-143.113,172.061,48.445,159.604
C04293=1024.695,364.082,-143.153,172.068,48.446,159.605
C04294=1024.704,364.329,-143.192,172.075,48.447,159.606
C04295=1024.711,364.575,-143.231,172.083,48.446,159.608
C04296=1024.720,364.822,-143.270,172.091,48.447,159.609
C04297=1024.728,365.069,-143.309,172.099,48.447,159.610
C04298=1024.736,365.315,-143.349,172.107,48.448,159.611
C04299=1024.744,365.548,-143.386,172.114,48.448,159.612
C04300=1024.752,365.781,-143.423,172.121,48.448,159.614
C04301=1024.760,366.014,-143.460,172.129,48.448,159.615
C04302=1024.767,366.246,-143.498,172.136,48.448,159.616
C04303=1024.776,366.479,-143.535,172.144,48.449,159.617
C04304=1024.783,366.711,-143.571,172.151,48.450,159.618
C04305=1024.791,366.944,-143.609,172.158,48.450,159.619
C04306=1024.798,367.176,-143.646,172.166,48.450,159.620
C04307=1024.807,367.423,-143.685,172.174,48.450,159.622
C04308=1024.815,367.670,-143.725,172.181,48.451,159.623
C04309=1024.824,367.917,-143.764,172.190,48.451,159.624
C04310=1024.832,368.164,-143.804,172.198,48.452,159.626
C04311=1024.841,368.410,-143.844,172.206,48.452,159.627
C04312=1024.849,368.656,-143.884,172.214,48.452,159.628
C04313=1024.857,368.903,-143.924,172.222,48.454,159.629
C04314=1024.866,369.149,-143.964,172.230,48.454,159.631
C04315=1024.874,369.397,-144.004,172.238,48.454,159.632
C04316=1024.883,369.644,-144.043,172.246,48.455,159.633
C04317=1024.891,369.890,-144.084,172.254,48.456,159.635
C04318=1024.898,370.137,-144.124,172.262,48.456,159.636
C04319=1024.907,370.383,-144.164,172.271,48.456,159.637
C04320=1024.915,370.630,-144.204,172.278,48.457,159.639
C04321=1024.924,370.876,-144.244,172.287,48.458,159.640
C04322=1024.932,371.123,-144.284,172.295,48.458,159.641
C04323=1024.941,371.369,-144.324,172.303,48.459,159.643
C04324=1024.949,371.616,-144.365,172.311,48.459,159.644
C04325=1024.958,371.863,-144.405,172.320,48.460,159.645
C04326=1024.966,372.109,-144.445,172.327,48.461,159.647
C04327=1024.974,372.356,-144.486,172.336,48.462,159.648
C04328=1024.983,372.603,-144.525,172.345,48.463,159.650
C04329=1024.991,372.849,-144.566,172.352,48.463,159.651
C04330=1025.000,373.096,-144.607,172.361,48.464,159.652
C04331=1025.008,373.342,-144.647,172.369,48.464,159.654
C04332=1025.018,373.589,-144.688,172.377,48.465,159.655
C04333=1025.026,373.835,-144.728,172.386,48.466,159.656
C04334=1025.035,374.082,-144.768,172.394,48.466,159.658
C04335=1025.043,374.328,-144.809,172.403,48.467,159.659
C04336=1025.051,374.575,-144.850,172.411,48.468,159.661
C04337=1025.060,374.821,-144.890,172.419,48.469,159.662
C04338=1025.069,375.068,-144.931,172.428,48.469,159.663
C04339=1025.078,375.314,-144.971,172.437,48.470,159.665
C04340=1025.086,375.561,-145.012,172.445,48.471,159.666
C04341=1025.095,375.807,-145.052,172.453,48.472,159.668
C04342=1025.104,376.054,-145.093,172.462,48.473,159.669
C04343=1025.113,376.300,-145.134,172.471,48.474,159.671
C04344=1025.121,376.547,-145.174,172.479,48.475,159.672
C04345=1025.130,376.794,-145.215,172.488,48.476,159.674
C04346=1025.138,377.041,-145.256,172.497,48.476,159.675
C04347=1025.148,377.286,-145.297,172.504,48.478,159.677
C04348=1025.156,377.533,-145.338,172.513,48.478,159.678
C04349=1025.165,377.779,-145.380,172.522,48.479,159.680
C04350=1025.173,378.026,-145.421,172.531,48.481,159.681
C04351=1025.182,378.272,-145.462,172.540,48.482,159.683
C04352=1025.190,378.518,-145.503,172.549,48.482,159.684
C04353=1025.199,378.765,-145.545,172.557,48.483,159.686
C04354=1025.208,379.011,-145.586,172.566,48.485,159.687
C04355=1025.217,379.258,-145.627,172.575,48.485,159.689
C04356=1025.225,379.504,-145.669,172.583,48.487,159.690
C04357=1025.235,379.750,-145.710,172.592,48.488,159.692
C04358=1025.243,379.997,-145.751,172.601,48.489,159.694
C04359=1025.252,380.239,-145.792,172.609,48.490,159.695
C04360=1025.261,380.483,-145.833,172.618,48.491,159.697
C04361=1025.269,380.727,-145.874,172.627,48.492,159.698
C04362=1025.279,380.970,-145.915,172.636,48.493,159.700
C04363=1025.287,381.213,-145.956,172.645,48.494,159.701
C04364=1025.295,381.456,-145.997,172.654,48.496,159.703
C04365=1025.305,381.699,-146.038,172.663,48.496,159.705
C04366=1025.313,381.943,-146.079,172.672,48.498,159.706
C04367=1025.322,382.190,-146.121,172.681,48.499,159.708
C04368=1025.331,382.435,-146.162,172.690,48.500,159.709
C04369=1025.340,382.682,-146.204,172.699,48.501,159.711
C04370=1025.349,382.928,-146.246,172.708,48.502,159.713
C04371=1025.358,383.174,-146.287,172.717,48.504,159.714
C04372=1025.367,383.421,-146.329,172.726,48.505,159.716
C04373=1025.376,383.667,-146.372,172.735,48.506,159.718
C04374=1025.385,383.914,-146.414,172.744,48.508,159.719
C04375=1025.395,384.160,-146.455,172.754,48.508,159.721
C04376=1025.404,384.406,-146.496,172.763,48.510,159.723
C04377=1025.413,384.652,-146.539,172.772,48.511,159.724
C04378=1025.422,384.898,-146.581,172.781,48.512,159.726
C04379=1025.431,385.144,-146.622,172.790,48.514,159.728
C04380=1025.440,385.390,-146.665,172.800,48.515,159.729
C04381=1025.450,385.637,-146.707,172.809,48.516,159.731
C04382=1025.459,385.884,-146.748,172.818,48.518,159.733
C04383=1025.468,386.129,-146.791,172.827,48.519,159.735
C04384=1025.477,386.375,-146.833,172.837,48.520,159.736
C04385=1025.487,386.622,-146.875,172.847,48.522,159.738
C04386=1025.496,386.868,-146.918,172.856,48.524,159.740
C04387=1025.505,387.114,-146.960,172.865,48.525,159.742
C04388=1025.513,387.360,-147.003,172.874,48.526,159.743
C04389=1025.523,387.607,-147.045,172.885,48.528,159.745
C04390=1025.532,387.852,-147.088,172.894,48.529,159.747
C04391=1025.542,388.098,-147.130,172.903,48.531,159.749
C04392=1025.552,388.345,-147.173,172.913,48.532,159.751
C04393=1025.560,388.591,-147.215,172.922,48.534,159.752
C04394=1025.569,388.837,-147.258,172.932,48.536,159.754
C04395=1025.579,389.084,-147.301,172.942,48.537,159.756
C04396=1025.588,389.329,-147.343,172.951,48.539,159.758
C04397=1025.597,389.576,-147.386,172.961,48.541,159.760
C04398=1025.607,389.821,-147.430,172.971,48.542,159.761
C04399=1025.617,390.068,-147.472,172.980,48.544,159.763
C04400=1025.625,390.314,-147.515,172.989,48.545,159.765
C04401=1025.635,390.560,-147.558,173.000,48.547,159.767
C04402=1025.644,390.806,-147.601,173.009,48.549,159.769
C04403=1025.654,391.052,-147.645,173.020,48.550,159.771
C04404=1025.663,391.298,-147.687,173.029,48.552,159.773
C04405=1025.673,391.544,-147.730,173.039,48.553,159.775
C04406=1025.681,391.790,-147.774,173.049,48.555,159.776
C04407=1025.691,392.036,-147.816,173.059,48.557,159.778
C04408=1025.701,392.282,-147.859,173.069,48.559,159.780
C04409=1025.710,392.528,-147.903,173.079,48.560,159.782
C04410=1025.720,392.774,-147.946,173.089,48.562,159.784
C04411=1025.729,393.019,-147.989,173.099,48.564,159.786
C04412=1025.739,393.266,-148.033,173.108,48.566,159.788
C04413=1025.749,393.512,-148.076,173.119,48.567,159.790
C04414=1025.758,393.758,-148.120,173.128,48.569,159.792
C04415=1025.768,394.003,-148.163,173.139,48.572,159.794
C04416=1025.777,394.250,-148.207,173.150,48.573,159.796
C04417=1025.787,394.496,-148.250,173.159,48.575,159.798
C04418=1025.796,394.742,-148.294,173.170,48.577,159.800
C04419=1025.810,395.091,-148.356,173.184,48.580,159.803
C04420=1025.824,395.440,-148.418,173.199,48.582,159.806
C04421=1025.837,395.789,-148.480,173.213,48.586,159.809
C04422=1025.851,396.139,-148.542,173.227,48.588,159.811
C04423=1025.861,396.385,-148.586,173.238,48.590,159.814
C04424=1025.871,396.631,-148.630,173.248,48.592,159.815
C04425=1025.880,396.877,-148.674,173.259,48.594,159.818
C04426=1025.891,397.122,-148.718,173.269,48.596,159.820
C04427=1025.900,397.368,-148.762,173.280,48.598,159.822
C04428=1025.910,397.614,-148.806,173.290,48.600,159.824
C04429=1025.919,397.860,-148.850,173.301,48.602,159.826
C04430=1025.930,398.105,-148.894,173.311,48.604,159.828
C04431=1025.939,398.351,-148.938,173.321,48.606,159.830
C04432=1025.949,398.597,-148.983,173.332,48.609,159.832
C04433=1025.959,398.843,-149.027,173.343,48.611,159.834
C04434=1025.969,399.089,-149.071,173.354,48.613,159.837
C04435=1025.978,399.334,-149.116,173.365,48.615,159.839
C04436=1025.989,399.580,-149.160,173.375,48.617,159.841
C04437=1025.999,399.826,-149.204,173.385,48.620,159.843
C04438=1026.009,400.072,-149.249,173.396,48.622,159.845
C04439=1026.018,400.318,-149.294,173.407,48.624,159.847
C04440=1026.029,400.563,-149.338,173.418,48.626,159.850
C04441=1026.039,400.810,-149.383,173.428,48.628,159.852
C04442=1026.048,401.055,-149.427,173.439,48.630,159.854
C04443=1026.057,401.264,-149.466,173.449,48.632,159.856
C04444=1026.065,401.474,-149.504,173.458,48.634,159.858
C04445=1026.074,401.683,-149.542,173.468,48.636,159.860
C04446=1026.083,401.893,-149.580,173.476,48.639,159.862
C04447=1026.091,402.102,-149.619,173.486,48.641,159.864
C04448=1026.100,402.312,-149.656,173.495,48.643,159.866
C04449=1026.108,402.521,-149.695,173.505,48.644,159.867
C04450=1026.117,402.731,-149.734,173.514,48.646,159.869
C04451=1026.126,402.976,-149.779,173.525,48.649,159.872
C04452=1026.137,403.222,-149.824,173.536,48.651,159.874
C04453=1026.146,403.468,-149.869,173.547,48.654,159.876
C04454=1026.156,403.713,-149.915,173.559,48.657,159.879
C04455=1026.167,403.959,-149.960,173.569,48.659,159.881
C04456=1026.177,404.204,-150.004,173.581,48.661,159.883
C04457=1026.188,404.450,-150.050,173.593,48.664,159.886
C04458=1026.198,404.696,-150.095,173.604,48.666,159.888
C04459=1026.208,404.941,-150.141,173.615,48.669,159.890
C04460=1026.219,405.187,-150.186,173.626,48.671,159.893
C04461=1026.229,405.432,-150.231,173.637,48.674,159.895
C04462=1026.239,405.678,-150.277,173.649,48.676,159.898
C04463=1026.250,405.924,-150.322,173.660,48.679,159.900
C04464=1026.260,406.169,-150.368,173.671,48.682,159.902
C04465=1026.270,406.415,-150.413,173.684,48.684,159.905
C04466=1026.280,406.661,-150.459,173.695,48.687,159.907
C04467=1026.291,406.906,-150.505,173.706,48.689,159.910
C04468=1026.301,407.151,-150.551,173.718,48.692,159.912
C04469=1026.312,407.397,-150.596,173.730,48.695,159.915
C04470=1026.322,407.642,-150.642,173.741,48.698,159.917
C04471=1026.333,407.888,-150.688,173.753,48.700,159.919
C04472=1026.343,408.134,-150.733,173.764,48.703,159.922
C04473=1026.354,408.380,-150.779,173.777,48.706,159.925
C04474=1026.365,408.625,-150.825,173.788,48.708,159.927
C04475=1026.375,408.870,-150.872,173.800,48.711,159.929
C04476=1026.386,409.116,-150.918,173.812,48.714,159.932
C04477=1026.397,409.361,-150.964,173.824,48.716,159.934
C04478=1026.407,409.607,-151.010,173.835,48.719,159.937
C04479=1026.421,409.905,-151.066,173.851,48.723,159.940
C04480=1026.433,410.205,-151.121,173.865,48.726,159.943
C04481=1026.446,410.504,-151.179,173.879,48.730,159.946
C04482=1026.460,410.803,-151.235,173.894,48.733,159.950
C04483=1026.470,411.048,-151.282,173.905,48.736,159.952
C04484=1026.480,411.294,-151.328,173.918,48.739,159.955
C04485=1026.491,411.539,-151.375,173.930,48.742,159.958
C04486=1026.503,411.784,-151.422,173.942,48.745,159.960
C04487=1026.513,412.030,-151.468,173.955,48.748,159.963
C04488=1026.524,412.275,-151.515,173.967,48.751,159.965
C04489=1026.535,412.520,-151.561,173.980,48.754,159.968
C04490=1026.545,412.766,-151.609,173.991,48.757,159.971
C04491=1026.556,413.011,-151.656,174.004,48.760,159.974
C04492=1026.567,413.256,-151.702,174.017,48.763,159.976
C04493=1026.579,413.502,-151.749,174.029,48.766,159.979
C04494=1026.589,413.747,-151.796,174.042,48.769,159.982
C04495=1026.600,413.993,-151.843,174.054,48.773,159.984
C04496=1026.611,414.238,-151.890,174.066,48.776,159.987
C04497=1026.622,414.483,-151.937,174.079,48.779,159.990
C04498=1026.633,414.729,-151.984,174.092,48.782,159.993
C04499=1026.645,414.974,-152.031,174.104,48.785,159.996
C04500=1026.655,415.220,-152.078,174.117,48.788,159.998
C04501=1026.667,415.465,-152.126,174.130,48.791,160.001
C04502=1026.678,415.710,-152.173,174.142,48.794,160.004
C04503=1026.689,415.955,-152.220,174.155,48.798,160.007
C04504=1026.700,416.201,-152.268,174.168,48.801,160.010
C04505=1026.712,416.445,-152.315,174.181,48.804,160.013
C04506=1026.722,416.691,-152.363,174.194,48.808,160.015
C04507=1026.733,416.936,-152.411,174.207,48.811,160.018
C04508=1026.745,417.181,-152.459,174.220,48.815,160.021
C04509=1026.755,417.427,-152.506,174.233,48.818,160.024
C04510=1026.767,417.672,-152.554,174.246,48.821,160.027
C04511=1026.778,417.916,-152.602,174.260,48.824,160.030
C04512=1026.790,418.161,-152.650,174.272,48.828,160.033
C04513=1026.801,418.407,-152.698,174.285,48.831,160.036
C04514=1026.812,418.652,-152.746,174.299,48.835,160.039
C04515=1026.824,418.897,-152.794,174.312,48.838,160.042
C04516=1026.835,419.143,-152.842,174.325,48.841,160.045
C04517=1026.847,419.388,-152.890,174.339,48.845,160.048
C04518=1026.858,419.633,-152.938,174.352,48.849,160.051
C04519=1026.869,419.878,-152.986,174.366,48.852,160.054
C04520=1026.881,420.123,-153.035,174.379,48.855,160.057
C04521=1026.893,420.368,-153.083,174.392,48.859,160.060
C04522=1026.904,420.613,-153.131,174.406,48.862,160.063
C04523=1026.915,420.858,-153.180,174.419,48.866,160.066
C04524=1026.927,421.103,-153.228,174.434,48.870,160.069
C04525=1026.938,421.348,-153.276,174.447,48.874,160.072
C04526=1026.950,421.593,-153.324,174.461,48.877,160.075
C04527=1026.962,421.839,-153.373,174.474,48.881,160.078
C04528=1026.974,422.083,-153.421,174.488,48.884,160.081
C04529=1026.986,422.328,-153.470,174.502,48.888,160.085
C04530=1026.997,422.573,-153.519,174.516,48.891,160.088
C04531=1027.009,422.819,-153.568,174.530,48.895,160.091
C04532=1027.021,423.063,-153.616,174.544,48.899,160.094
C04533=1027.032,423.308,-153.666,174.558,48.903,160.097
C04534=1027.044,423.553,-153.715,174.572,48.906,160.101
C04535=1027.056,423.798,-153.764,174.586,48.911,160.104
C04536=1027.067,424.043,-153.813,174.600,48.914,160.107
C04537=1027.080,424.288,-153.862,174.615,48.918,160.110
C04538=1027.091,424.533,-153.911,174.629,48.922,160.114
C04539=1027.106,424.842,-153.973,174.647,48.927,160.118
C04540=1027.122,425.152,-154.035,174.665,48.932,160.122
C04541=1027.137,425.462,-154.098,174.683,48.937,160.126
C04542=1027.151,425.771,-154.160,174.701,48.942,160.130
C04543=1027.164,426.016,-154.210,174.716,48.946,160.134
C04544=1027.176,426.261,-154.259,174.730,48.949,160.137
C04545=1027.188,426.505,-154.309,174.745,48.953,160.140
C04546=1027.200,426.750,-154.359,174.759,48.957,160.144
C04547=1027.212,426.996,-154.408,174.774,48.962,160.147
C04548=1027.224,427.240,-154.458,174.789,48.966,160.151
C04549=1027.236,427.484,-154.508,174.804,48.970,160.154
C04550=1027.249,427.729,-154.558,174.819,48.974,160.158
C04551=1027.261,427.974,-154.608,174.834,48.978,160.161
C04552=1027.273,428.218,-154.658,174.849,48.982,160.165
C04553=1027.285,428.463,-154.708,174.864,48.986,160.168
C04554=1027.297,428.708,-154.758,174.879,48.991,160.172
C04555=1027.309,428.953,-154.809,174.893,48.995,160.175
C04556=1027.321,429.198,-154.859,174.909,48.999,160.179
C04557=1027.334,429.442,-154.910,174.924,49.003,160.182
C04558=1027.346,429.687,-154.960,174.939,49.007,160.186
C04559=1027.359,429.932,-155.010,174.955,49.012,160.190
C04560=1027.371,430.176,-155.061,174.970,49.016,160.193
C04561=1027.384,430.421,-155.111,174.986,49.020,160.197
C04562=1027.396,430.665,-155.162,175.001,49.024,160.200
C04563=1027.408,430.910,-155.212,175.016,49.029,160.204
C04564=1027.422,431.155,-155.263,175.032,49.033,160.208
C04565=1027.434,431.399,-155.314,175.047,49.037,160.211
C04566=1027.447,431.644,-155.364,175.063,49.042,160.215
C04567=1027.459,431.888,-155.415,175.079,49.046,160.219
C04568=1027.472,432.133,-155.466,175.095,49.051,160.222
C04569=1027.485,432.377,-155.517,175.111,49.055,160.226
C04570=1027.498,432.621,-155.568,175.127,49.059,160.230
C04571=1027.511,432.866,-155.619,175.142,49.064,160.234
C04572=1027.524,433.110,-155.670,175.158,49.068,160.237
C04573=1027.537,433.355,-155.721,175.174,49.073,160.241
C04574=1027.549,433.599,-155.772,175.191,49.077,160.245
C04575=1027.563,433.844,-155.823,175.206,49.082,160.249
C04576=1027.576,434.088,-155.874,175.222,49.086,160.253
C04577=1027.588,434.333,-155.926,175.239,49.091,160.257
C04578=1027.601,434.577,-155.977,175.255,49.096,160.261
C04579=1027.614,434.822,-156.029,175.272,49.100,160.264
C04580=1027.627,435.066,-156.080,175.288,49.105,160.268
C04581=1027.640,435.310,-156.131,175.304,49.110,160.272
C04582=1027.653,435.555,-156.184,175.321,49.114,160.276
C04583=1027.666,435.799,-156.235,175.337,49.119,160.280
C04584=1027.679,436.043,-156.287,175.354,49.124,160.284
C04585=1027.692,436.288,-156.339,175.370,49.129,160.288
C04586=1027.706,436.532,-156.391,175.388,49.133,160.292
C04587=1027.718,436.776,-156.443,175.405,49.138,160.296
C04588=1027.732,437.020,-156.494,175.421,49.142,160.300
C04589=1027.745,437.264,-156.547,175.438,49.148,160.304
C04590=1027.758,437.509,-156.599,175.456,49.152,160.309
C04591=1027.772,437.752,-156.651,175.472,49.157,160.312
C04592=1027.785,437.997,-156.704,175.489,49.162,160.317
C04593=1027.798,438.241,-156.756,175.507,49.167,160.321
C04594=1027.812,438.485,-156.808,175.524,49.172,160.325
C04595=1027.825,438.729,-156.861,175.541,49.177,160.329
C04596=1027.839,438.973,-156.914,175.558,49.182,160.333
C04597=1027.852,439.217,-156.965,175.576,49.186,160.337
C04598=1027.866,439.461,-157.019,175.593,49.192,160.342
C04599=1027.879,439.709,-157.072,175.611,49.197,160.346
C04600=1027.893,439.957,-157.126,175.629,49.202,160.350
C04601=1027.907,440.205,-157.179,175.647,49.207,160.355
C04602=1027.921,440.452,-157.233,175.664,49.212,160.359
C04603=1027.935,440.697,-157.287,175.682,49.217,160.363
C04604=1027.949,440.940,-157.339,175.700,49.223,160.368
C04605=1027.962,441.184,-157.392,175.718,49.227,160.372
C04606=1027.976,441.429,-157.445,175.736,49.232,160.377
C04607=1027.990,441.672,-157.498,175.755,49.238,160.381
C04608=1028.004,441.917,-157.552,175.773,49.243,160.385
C04609=1028.018,442.160,-157.605,175.791,49.248,160.390
C04610=1028.032,442.405,-157.658,175.809,49.253,160.394
C04611=1028.045,442.647,-157.711,175.827,49.258,160.399
C04612=1028.060,442.890,-157.764,175.846,49.263,160.403
C04613=1028.075,443.134,-157.817,175.864,49.269,160.408
C04614=1028.089,443.377,-157.870,175.882,49.274,160.412
C04615=1028.105,443.620,-157.922,175.900,49.279,160.416
C04616=1028.121,443.863,-157.973,175.919,49.284,160.421
C04617=1028.138,444.108,-158.025,175.938,49.288,160.425
C04618=1028.154,444.352,-158.075,175.957,49.293,160.430
C04619=1028.172,444.595,-158.126,175.976,49.298,160.434
C04620=1028.189,444.839,-158.176,175.995,49.303,160.439
C04621=1028.208,445.083,-158.226,176.014,49.308,160.443
C04622=1028.227,445.327,-158.275,176.033,49.312,160.448
C04623=1028.246,445.571,-158.324,176.052,49.316,160.452
C04624=1028.266,445.815,-158.371,176.072,49.321,160.457
C04625=1028.286,446.059,-158.420,176.091,49.325,160.461
C04626=1028.306,446.303,-158.468,176.111,49.329,160.465
C04627=1028.327,446.548,-158.515,176.130,49.333,160.470
C04628=1028.349,446.792,-158.562,176.150,49.338,160.474
C04629=1028.371,447.037,-158.608,176.170,49.341,160.478
C04630=1028.393,447.282,-158.654,176.190,49.345,160.483
C04631=1028.417,447.526,-158.700,176.210,49.349,160.487
C04632=1028.440,447.771,-158.745,176.229,49.353,160.491
C04633=1028.464,448.016,-158.790,176.249,49.357,160.496
C04634=1028.488,448.261,-158.834,176.270,49.360,160.500
C04635=1028.513,448.505,-158.879,176.290,49.364,160.505
C04636=1028.539,448.751,-158.922,176.310,49.367,160.509
C04637=1028.565,448.996,-158.966,176.331,49.371,160.513
C04638=1028.591,449.240,-159.008,176.351,49.375,160.518
C04639=1028.618,449.486,-159.051,176.372,49.378,160.522
C04640=1028.645,449.731,-159.092,176.393,49.381,160.526
C04641=1028.672,449.976,-159.134,176.413,49.385,160.531
C04642=1028.701,450.222,-159.175,176.435,49.387,160.535
C04643=1028.729,450.467,-159.217,176.456,49.391,160.539
C04644=1028.759,450.713,-159.257,176.476,49.394,160.544
C04645=1028.788,450.958,-159.297,176.498,49.397,160.548
C04646=1028.818,451.203,-159.337,176.519,49.399,160.552
C04647=1028.848,451.448,-159.376,176.540,49.403,160.557
C04648=1028.880,451.694,-159.415,176.562,49.405,160.561
C04649=1028.911,451.940,-159.453,176.583,49.408,160.565
C04650=1028.943,452.185,-159.491,176.605,49.410,160.569
C04651=1028.976,452.431,-159.529,176.626,49.413,160.574
C04652=1029.008,452.677,-159.566,176.649,49.416,160.578
C04653=1029.042,452.922,-159.603,176.670,49.418,160.582
C04654=1029.075,453.168,-159.639,176.692,49.421,160.587
C04655=1029.110,453.414,-159.675,176.715,49.423,160.591
C04656=1029.145,453.660,-159.711,176.737,49.425,160.595
C04657=1029.180,453.905,-159.746,176.759,49.428,160.600
C04658=1029.216,454.151,-159.781,176.781,49.430,160.604
C04659=1028.939,454.225,-160.117,176.784,49.492,160.624
C04660=1028.903,453.979,-160.082,176.762,49.489,160.620
C04661=1028.868,453.733,-160.047,176.739,49.487,160.615
C04662=1028.833,453.488,-160.011,176.717,49.485,160.611
C04663=1028.798,453.241,-159.975,176.695,49.483,160.607
C04664=1028.765,452.996,-159.939,176.673,49.480,160.602
C04665=1028.731,452.751,-159.902,176.651,49.478,160.598
C04666=1028.697,452.505,-159.866,176.629,49.476,160.594
C04667=1028.665,452.259,-159.828,176.607,49.473,160.589
C04668=1028.633,452.014,-159.790,176.586,49.470,160.585
C04669=1028.601,451.769,-159.752,176.564,49.467,160.581
C04670=1028.570,451.523,-159.713,176.543,49.465,160.577
C04671=1028.539,451.277,-159.674,176.521,49.462,160.572
C04672=1028.510,451.032,-159.634,176.499,49.460,160.568
C04673=1028.480,450.786,-159.595,176.479,49.456,160.564
C04674=1028.451,450.540,-159.554,176.457,49.454,160.559
C04675=1028.422,450.295,-159.514,176.436,49.450,160.555
C04676=1028.393,450.049,-159.473,176.415,49.448,160.551
C04677=1028.365,449.805,-159.431,176.394,49.444,160.546
C04678=1028.339,449.559,-159.389,176.373,49.441,160.542
C04679=1028.310,449.314,-159.347,176.353,49.438,160.538
C04680=1028.284,449.069,-159.304,176.332,49.435,160.533
C04681=1028.258,448.824,-159.261,176.311,49.431,160.529
C04682=1028.233,448.579,-159.218,176.291,49.428,160.525
C04683=1028.208,448.334,-159.175,176.271,49.425,160.520
C04684=1028.183,448.089,-159.129,176.250,49.421,160.516
C04685=1028.159,447.844,-159.085,176.230,49.418,160.512
C04686=1028.136,447.599,-159.039,176.210,49.413,160.507
C04687=1028.113,447.355,-158.994,176.190,49.410,160.503
C04688=1028.090,447.110,-158.948,176.171,49.406,160.499
C04689=1028.068,446.866,-158.902,176.151,49.402,160.494
C04690=1028.046,446.621,-158.855,176.131,49.398,160.490
C04691=1028.025,446.377,-158.809,176.111,49.394,160.485
C04692=1028.004,446.133,-158.761,176.091,49.391,160.481
C04693=1027.983,445.888,-158.713,176.072,49.386,160.477
C04694=1027.964,445.644,-158.665,176.052,49.382,160.472
C04695=1027.944,445.400,-158.617,176.033,49.378,160.468
C04696=1027.925,445.155,-158.567,176.014,49.373,160.463
C04697=1027.906,444.911,-158.518,175.995,49.369,160.459
C04698=1027.889,444.668,-158.468,175.976,49.364,160.455
C04699=1027.870,444.424,-158.418,175.957,49.360,160.450
C04700=1027.854,444.180,-158.367,175.938,49.355,160.446
C04701=1027.837,443.937,-158.316,175.919,49.350,160.441
C04702=1027.820,443.693,-158.265,175.901,49.345,160.437
C04703=1027.804,443.450,-158.213,175.881,49.341,160.432
C04704=1027.790,443.206,-158.161,175.863,49.336,160.428
C04705=1027.774,442.963,-158.108,175.844,49.331,160.423
C04706=1027.760,442.719,-158.055,175.826,49.326,160.419
C04707=1027.746,442.476,-158.002,175.808,49.321,160.415
C04708=1027.732,442.233,-157.949,175.790,49.316,160.410
C04709=1027.718,441.988,-157.895,175.772,49.311,160.406
C04710=1027.705,441.745,-157.843,175.753,49.306,160.401
C04711=1027.691,441.502,-157.789,175.735,49.300,160.397
C04712=1027.677,441.260,-157.736,175.717,49.295,160.392
C04713=1027.663,441.019,-157.684,175.699,49.291,160.388
C04714=1027.649,440.778,-157.632,175.682,49.286,160.384
C04715=1027.636,440.536,-157.579,175.664,49.280,160.380
C04716=1027.623,440.295,-157.527,175.646,49.276,160.375
C04717=1027.609,440.053,-157.475,175.629,49.271,160.371
C04718=1027.595,439.812,-157.423,175.612,49.266,160.367
C04719=1027.582,439.570,-157.370,175.595,49.261,160.363
C04720=1027.569,439.327,-157.318,175.577,49.256,160.359
C04721=1027.555,439.083,-157.265,175.559,49.251,160.354
C04722=1027.542,438.839,-157.213,175.542,49.246,160.350
C04723=1027.528,438.595,-157.160,175.524,49.241,160.346
C04724=1027.515,438.350,-157.108,175.508,49.237,160.342
C04725=1027.501,438.106,-157.055,175.490,49.232,160.338
C04726=1027.487,437.862,-157.003,175.473,49.227,160.333
C04727=1027.475,437.617,-156.950,175.455,49.222,160.329
C04728=1027.461,437.373,-156.898,175.439,49.218,160.325
C04729=1027.448,437.129,-156.847,175.422,49.213,160.321
C04730=1027.434,436.886,-156.794,175.404,49.208,160.317
C04731=1027.421,436.641,-156.742,175.388,49.203,160.313
C04732=1027.408,436.397,-156.690,175.371,49.199,160.309
C04733=1027.395,436.152,-156.639,175.355,49.194,160.305
C04734=1027.383,435.908,-156.586,175.337,49.190,160.301
C04735=1027.369,435.664,-156.535,175.320,49.185,160.297
C04736=1027.355,435.419,-156.483,175.304,49.180,160.293
C04737=1027.343,435.175,-156.432,175.288,49.176,160.289
C04738=1027.330,434.931,-156.379,175.271,49.171,160.285
C04739=1027.317,434.686,-156.328,175.255,49.166,160.281
C04740=1027.304,434.442,-156.277,175.239,49.162,160.278
C04741=1027.291,434.197,-156.226,175.222,49.158,160.274
C04742=1027.278,433.954,-156.174,175.206,49.153,160.270
C04743=1027.265,433.708,-156.122,175.190,49.149,160.266
C04744=1027.253,433.464,-156.071,175.173,49.144,160.262
C04745=1027.239,433.220,-156.020,175.158,49.139,160.258
C04746=1027.227,432.976,-155.969,175.142,49.135,160.255
C04747=1027.213,432.731,-155.918,175.126,49.131,160.251
C04748=1027.201,432.486,-155.867,175.109,49.127,160.247
C04749=1027.188,432.242,-155.817,175.094,49.122,160.243
C04750=1027.175,431.997,-155.765,175.078,49.118,160.240
C04751=1027.163,431.753,-155.715,175.062,49.114,160.236
C04752=1027.150,431.508,-155.664,175.047,49.109,160.232
C04753=1027.137,431.263,-155.613,175.031,49.105,160.229
C04754=1027.124,431.019,-155.563,175.015,49.101,160.225
C04755=1027.112,430.775,-155.512,175.000,49.097,160.221
C04756=1027.099,430.530,-155.462,174.984,49.093,160.217
C04757=1027.087,430.286,-155.411,174.969,49.088,160.214
C04758=1027.075,430.041,-155.361,174.953,49.084,160.210
C04759=1027.062,429.797,-155.310,174.938,49.080,160.207
C04760=1027.050,429.552,-155.260,174.922,49.076,160.203
C04761=1027.037,429.307,-155.210,174.907,49.072,160.200
C04762=1027.025,429.062,-155.160,174.892,49.068,160.196
C04763=1027.012,428.818,-155.109,174.876,49.064,160.192
C04764=1027.000,428.573,-155.059,174.862,49.060,160.189
C04765=1026.988,428.328,-155.009,174.847,49.055,160.185
C04766=1026.975,428.083,-154.959,174.832,49.051,160.182
C04767=1026.964,427.839,-154.909,174.816,49.048,160.179
C04768=1026.951,427.594,-154.859,174.802,49.044,160.175
C04769=1026.939,427.350,-154.809,174.787,49.040,160.172
C04770=1026.927,427.104,-154.759,174.772,49.036,160.168
C04771=1026.915,426.860,-154.710,174.758,49.032,160.165
C04772=1026.903,426.615,-154.659,174.743,49.028,160.161
C04773=1026.891,426.370,-154.609,174.728,49.024,160.158
C04774=1026.879,426.126,-154.560,174.714,49.020,160.155
C04775=1026.867,425.881,-154.510,174.699,49.016,160.151
C04776=1026.851,425.569,-154.448,174.680,49.011,160.147
C04777=1026.836,425.257,-154.384,174.661,49.006,160.143
C04778=1026.820,424.945,-154.322,174.644,49.001,160.139
C04779=1026.806,424.633,-154.259,174.625,48.996,160.134
C04780=1026.794,424.389,-154.210,174.611,48.993,160.131
C04781=1026.781,424.143,-154.161,174.597,48.988,160.128
C04782=1026.770,423.899,-154.112,174.583,48.985,160.125
C04783=1026.758,423.653,-154.063,174.568,48.981,160.121
C04784=1026.747,423.408,-154.014,174.554,48.978,160.118
C04785=1026.735,423.164,-153.965,174.540,48.974,160.115
C04786=1026.722,422.919,-153.916,174.526,48.970,160.112
C04787=1026.711,422.674,-153.867,174.512,48.967,160.108
C04788=1026.700,422.429,-153.818,174.497,48.963,160.105
C04789=1026.688,422.184,-153.769,174.484,48.959,160.102
C04790=1026.676,421.939,-153.721,174.470,48.956,160.099
C04791=1026.665,421.693,-153.672,174.457,48.952,160.096
C04792=1026.652,421.449,-153.624,174.443,48.949,160.093
C04793=1026.641,421.203,-153.576,174.428,48.945,160.090
C04794=1026.629,420.959,-153.527,174.415,48.942,160.087
C04795=1026.618,420.713,-153.479,174.401,48.938,160.084
C04796=1026.606,420.468,-153.430,174.388,48.935,160.080
C04797=1026.594,420.223,-153.382,174.375,48.931,160.078
C04798=1026.583,419.978,-153.334,174.361,48.928,160.074
C04799=1026.571,419.733,-153.286,174.348,48.924,160.071
C04800=1026.560,419.487,-153.238,174.334,48.921,160.068
C04801=1026.548,419.242,-153.190,174.320,48.917,160.065
C04802=1026.537,418.998,-153.141,174.307,48.914,160.062
C04803=1026.526,418.753,-153.094,174.294,48.911,160.059
C04804=1026.515,418.508,-153.045,174.281,48.908,160.057
C04805=1026.504,418.263,-152.997,174.267,48.904,160.053
C04806=1026.492,418.017,-152.950,174.253,48.901,160.050
C04807=1026.481,417.771,-152.902,174.241,48.897,160.048
C04808=1026.470,417.527,-152.854,174.228,48.894,160.045
C04809=1026.459,417.282,-152.806,174.215,48.891,160.042
C04810=1026.447,417.037,-152.758,174.202,48.887,160.039
C04811=1026.436,416.791,-152.711,174.189,48.885,160.036
C04812=1026.425,416.546,-152.663,174.175,48.882,160.033
C04813=1026.414,416.301,-152.615,174.162,48.878,160.030
C04814=1026.403,416.056,-152.568,174.149,48.875,160.027
C04815=1026.392,415.811,-152.520,174.137,48.872,160.025
C04816=1026.380,415.565,-152.473,174.124,48.869,160.022
C04817=1026.369,415.320,-152.427,174.111,48.865,160.019
C04818=1026.358,415.074,-152.379,174.098,48.862,160.016
C04819=1026.347,414.829,-152.331,174.086,48.859,160.013
C04820=1026.336,414.584,-152.285,174.073,48.856,160.011
C04821=1026.325,414.339,-152.237,174.060,48.853,160.008
C04822=1026.314,414.093,-152.190,174.048,48.850,160.005
C04823=1026.303,413.848,-152.144,174.035,48.847,160.002
C04824=1026.291,413.602,-152.097,174.022,48.844,160.000
C04825=1026.281,413.357,-152.050,174.011,48.841,159.997
C04826=1026.270,413.111,-152.003,173.998,48.838,159.994
C04827=1026.259,412.866,-151.956,173.985,48.835,159.991
C04828=1026.249,412.621,-151.909,173.973,48.832,159.989
C04829=1026.238,412.376,-151.862,173.960,48.829,159.986
C04830=1026.226,412.131,-151.815,173.948,48.826,159.983
C04831=1026.215,411.885,-151.769,173.936,48.823,159.981
C04832=1026.205,411.640,-151.722,173.924,48.820,159.978
C04833=1026.194,411.395,-151.675,173.911,48.818,159.976
C04834=1026.183,411.148,-151.629,173.900,48.815,159.973
C04835=1026.172,410.903,-151.583,173.887,48.812,159.970
C04836=1026.160,410.602,-151.525,173.872,48.809,159.967
C04837=1026.147,410.301,-151.469,173.858,48.805,159.964
C04838=1026.134,410.000,-151.411,173.843,48.802,159.961
C04839=1026.121,409.699,-151.354,173.829,48.798,159.958
C04840=1026.110,409.453,-151.309,173.816,48.796,159.955
C04841=1026.099,409.207,-151.262,173.804,48.793,159.953
C04842=1026.088,408.961,-151.216,173.792,48.790,159.950
C04843=1026.078,408.716,-151.170,173.780,48.788,159.948
C04844=1026.068,408.471,-151.125,173.769,48.785,159.945
C04845=1026.057,408.225,-151.079,173.756,48.782,159.942
C04846=1026.046,407.979,-151.033,173.745,48.779,159.940
C04847=1026.036,407.734,-150.987,173.733,48.777,159.938
C04848=1026.025,407.488,-150.941,173.722,48.775,159.935
C04849=1026.014,407.243,-150.895,173.710,48.772,159.933
C04850=1026.004,406.997,-150.850,173.699,48.770,159.930
C04851=1025.992,406.752,-150.804,173.687,48.767,159.928
C04852=1025.983,406.506,-150.759,173.675,48.765,159.925
C04853=1025.972,406.261,-150.713,173.664,48.762,159.923
C04854=1025.962,406.015,-150.668,173.652,48.760,159.921
C04855=1025.952,405.770,-150.623,173.641,48.757,159.918
C04856=1025.941,405.524,-150.577,173.629,48.754,159.916
C04857=1025.931,405.278,-150.531,173.617,48.752,159.913
C04858=1025.921,405.033,-150.486,173.606,48.750,159.911
C04859=1025.910,404.787,-150.440,173.595,48.747,159.909
C04860=1025.900,404.541,-150.395,173.584,48.744,159.906
C04861=1025.890,404.296,-150.350,173.572,48.742,159.904
C04862=1025.880,404.050,-150.304,173.561,48.740,159.902
C04863=1025.870,403.804,-150.259,173.550,48.737,159.899
C04864=1025.859,403.559,-150.214,173.539,48.735,159.897
C04865=1025.850,403.313,-150.169,173.528,48.732,159.895
C04866=1025.840,403.068,-150.124,173.517,48.730,159.892
C04867=1025.829,402.822,-150.079,173.505,48.728,159.890
C04868=1025.819,402.576,-150.034,173.494,48.726,159.888
C04869=1025.808,402.331,-149.989,173.483,48.723,159.885
C04870=1025.799,402.085,-149.944,173.472,48.721,159.883
C04871=1025.789,401.840,-149.899,173.461,48.719,159.881
C04872=1025.779,401.594,-149.854,173.450,48.717,159.879
C04873=1025.769,401.348,-149.809,173.439,48.714,159.876
C04874=1025.759,401.103,-149.764,173.428,48.712,159.874
C04875=1025.750,400.856,-149.720,173.418,48.710,159.872
C04876=1025.739,400.611,-149.675,173.407,48.708,159.870
C04877=1025.729,400.365,-149.631,173.396,48.705,159.868
C04878=1025.719,400.120,-149.586,173.385,48.703,159.866
C04879=1025.710,399.873,-149.542,173.374,48.701,159.863
C04880=1025.699,399.628,-149.497,173.363,48.699,159.861
C04881=1025.689,399.382,-149.452,173.353,48.697,159.859
C04882=1025.680,399.136,-149.408,173.342,48.695,159.857
C04883=1025.669,398.891,-149.364,173.331,48.693,159.855
C04884=1025.660,398.644,-149.320,173.321,48.691,159.853
C04885=1025.650,398.399,-149.275,173.310,48.689,159.850
C04886=1025.640,398.153,-149.231,173.300,48.686,159.848
C04887=1025.631,397.907,-149.187,173.289,48.685,159.846
C04888=1025.620,397.662,-149.143,173.279,48.683,159.844
C04889=1025.611,397.416,-149.099,173.268,48.681,159.842
C04890=1025.601,397.170,-149.055,173.257,48.679,159.840
C04891=1025.591,396.924,-149.011,173.247,48.677,159.838
C04892=1025.581,396.678,-148.967,173.237,48.675,159.836
C04893=1025.571,396.432,-148.923,173.226,48.673,159.834
C04894=1025.562,396.186,-148.879,173.216,48.671,159.832
C04895=1025.552,395.940,-148.835,173.205,48.670,159.830
C04896=1025.541,395.662,-148.785,173.193,48.667,159.827
C04897=1025.530,395.382,-148.736,173.182,48.665,159.825
C04898=1025.519,395.103,-148.687,173.171,48.663,159.823
C04899=1025.508,394.825,-148.637,173.158,48.661,159.820
C04900=1025.499,394.578,-148.593,173.149,48.659,159.819
C04901=1025.489,394.333,-148.550,173.138,48.657,159.817
C04902=1025.480,394.086,-148.506,173.128,48.655,159.815
C04903=1025.470,393.841,-148.463,173.119,48.654,159.813
C04904=1025.461,393.595,-148.419,173.108,48.652,159.811
C04905=1025.451,393.348,-148.376,173.098,48.650,159.809
C04906=1025.441,393.102,-148.332,173.088,48.648,159.807
C04907=1025.432,392.857,-148.289,173.078,48.647,159.805
C04908=1025.422,392.610,-148.246,173.068,48.645,159.803
C04909=1025.413,392.364,-148.202,173.058,48.643,159.801
C04910=1025.403,392.119,-148.160,173.047,48.642,159.799
C04911=1025.393,391.872,-148.117,173.038,48.640,159.797
C04912=1025.385,391.627,-148.073,173.027,48.638,159.795
C04913=1025.375,391.380,-148.030,173.018,48.637,159.793
C04914=1025.365,391.134,-147.987,173.008,48.635,159.791
C04915=1025.356,390.888,-147.944,172.998,48.633,159.790
C04916=1025.341,390.506,-147.877,172.983,48.631,159.787
C04917=1025.327,390.123,-147.811,172.968,48.629,159.784
C04918=1025.313,389.741,-147.744,172.952,48.626,159.781
C04919=1025.298,389.359,-147.677,172.937,48.624,159.778
C04920=1025.289,389.113,-147.634,172.928,48.622,159.776
C04921=1025.279,388.867,-147.592,172.918,48.620,159.774
C04922=1025.270,388.620,-147.549,172.908,48.619,159.773
C04923=1025.261,388.374,-147.507,172.899,48.618,159.771
C04924=1025.252,388.128,-147.464,172.890,48.616,159.769
C04925=1025.242,387.881,-147.421,172.880,48.615,159.767
C04926=1025.233,387.636,-147.379,172.871,48.614,159.765
C04927=1025.224,387.390,-147.336,172.860,48.613,159.764
C04928=1025.214,387.143,-147.294,172.851,48.611,159.762
C04929=1025.205,386.897,-147.252,172.842,48.609,159.760
C04930=1025.196,386.651,-147.209,172.833,48.608,159.758
C04931=1025.188,386.405,-147.167,172.823,48.607,159.757
C04932=1025.178,386.158,-147.124,172.814,48.605,159.755
C04933=1025.169,385.912,-147.083,172.804,48.604,159.753
C04934=1025.160,385.666,-147.040,172.794,48.603,159.751
C04935=1025.151,385.420,-146.998,172.785,48.602,159.750
C04936=1025.141,385.174,-146.956,172.776,48.600,159.748
C04937=1025.132,384.927,-146.914,172.767,48.599,159.746
C04938=1025.122,384.681,-146.873,172.757,48.598,159.745
C04939=1025.113,384.435,-146.831,172.748,48.596,159.743
C04940=1025.104,384.189,-146.789,172.739,48.596,159.741
C04941=1025.095,383.943,-146.747,172.730,48.594,159.740
C04942=1025.086,383.696,-146.705,172.721,48.593,159.738
C04943=1025.077,383.450,-146.663,172.711,48.592,159.736
C04944=1025.068,383.203,-146.622,172.702,48.591,159.735
C04945=1025.059,382.957,-146.580,172.693,48.590,159.733
C04946=1025.050,382.711,-146.538,172.684,48.588,159.731
C04947=1025.041,382.465,-146.496,172.675,48.587,159.730
C04948=1025.032,382.219,-146.454,172.666,48.586,159.728
C04949=1025.023,381.973,-146.413,172.657,48.585,159.727
C04950=1025.014,381.726,-146.371,172.647,48.584,159.725
C04951=1025.005,381.479,-146.330,172.638,48.583,159.723
C04952=1024.992,381.127,-146.271,172.626,48.582,159.721
C04953=1024.980,380.775,-146.211,172.613,48.580,159.719
C04954=1024.967,380.422,-146.152,172.600,48.578,159.716
C04955=1024.955,380.071,-146.092,172.588,48.577,159.714
C04956=1024.946,379.824,-146.051,172.578,48.576,159.713
C04957=1024.937,379.577,-146.010,172.570,48.575,159.711
C04958=1024.928,379.331,-145.968,172.561,48.574,159.710
C04959=1024.919,379.085,-145.928,172.552,48.573,159.708
C04960=1024.910,378.839,-145.886,172.543,48.572,159.707
C04961=1024.902,378.592,-145.845,172.534,48.571,159.705
C04962=1024.893,378.345,-145.803,172.526,48.570,159.704
C04963=1024.884,378.100,-145.762,172.517,48.570,159.702
C04964=1024.876,377.853,-145.721,172.508,48.569,159.701
C04965=1024.867,377.606,-145.679,172.499,48.568,159.699
C04966=1024.859,377.360,-145.639,172.492,48.567,159.698
C04967=1024.850,377.113,-145.598,172.482,48.565,159.696
C04968=1024.842,376.867,-145.556,172.474,48.565,159.694
C04969=1024.833,376.621,-145.516,172.465,48.564,159.693
C04970=1024.824,376.374,-145.475,172.457,48.564,159.692
C04971=1024.815,376.128,-145.435,172.448,48.563,159.690
C04972=1024.807,375.881,-145.394,172.439,48.562,159.689
C04973=1024.798,375.634,-145.353,172.430,48.561,159.687
C04974=1024.789,375.388,-145.312,172.422,48.560,159.686
C04975=1024.780,375.141,-145.271,172.414,48.560,159.684
C04976=1024.771,374.895,-145.231,172.405,48.559,159.683
C04977=1024.763,374.648,-145.190,172.397,48.558,159.681
C04978=1024.754,374.402,-145.150,172.388,48.558,159.680
C04979=1024.746,374.155,-145.110,172.379,48.557,159.679
C04980=1024.737,373.909,-145.070,172.371,48.556,159.677
C04981=1024.728,373.662,-145.029,172.363,48.556,159.676
C04982=1024.720,373.416,-144.988,172.355,48.555,159.674
C04983=1024.712,373.170,-144.948,172.346,48.555,159.673
C04984=1024.703,372.923,-144.907,172.337,48.554,159.672
C04985=1024.694,372.676,-144.868,172.330,48.553,159.670
C04986=1024.686,372.429,-144.827,172.321,48.552,159.669
C04987=1024.677,372.183,-144.787,172.313,48.552,159.668
C04988=1024.669,371.937,-144.746,172.304,48.551,159.666
C04989=1024.660,371.690,-144.706,172.297,48.551,159.665
C04990=1024.652,371.443,-144.666,172.288,48.550,159.663
C04991=1024.643,371.197,-144.626,172.280,48.550,159.662
C04992=1024.635,370.950,-144.585,172.271,48.549,159.661
C04993=1024.627,370.703,-144.545,172.263,48.548,159.659
C04994=1024.618,370.457,-144.505,172.255,48.548,159.658
C04995=1024.610,370.210,-144.465,172.247,48.548,159.657
C04996=1024.602,369.964,-144.426,172.239,48.547,159.656
C04997=1024.594,369.716,-144.385,172.230,48.546,159.654
C04998=1024.585,369.470,-144.345,172.223,48.546,159.653
C04999=1024.577,369.223,-144.305,172.215,48.546,159.652
C05000=1024.568,368.977,-144.265,172.206,48.545,159.650
C05001=1024.561,368.731,-144.225,172.199,48.545,159.649
C05002=1024.552,368.484,-144.186,172.190,48.544,159.648
C05003=1024.544,368.236,-144.146,172.182,48.544,159.646
C05004=1024.535,367.990,-144.106,172.175,48.544,159.645
C05005=1024.527,367.744,-144.066,172.166,48.543,159.644
C05006=1024.518,367.497,-144.027,172.159,48.543,159.643
C05007=1024.510,367.250,-143.987,172.150,48.543,159.641
C05008=1024.502,367.016,-143.950,172.143,48.542,159.640
C05009=1024.494,366.783,-143.912,172.135,48.542,159.639
C05010=1024.487,366.549,-143.876,172.128,48.542,159.638
C05011=1024.478,366.316,-143.838,172.120,48.541,159.637
C05012=1024.470,366.082,-143.801,172.113,48.541,159.636
C05013=1024.463,365.848,-143.763,172.106,48.541,159.634
C05014=1024.455,365.614,-143.726,172.097,48.540,159.633
C05015=1024.447,365.381,-143.689,172.090,48.541,159.632
C05016=1024.439,365.134,-143.650,172.083,48.540,159.631
C05017=1024.430,364.887,-143.611,172.074,48.540,159.630
C05018=1024.423,364.640,-143.571,172.067,48.540,159.629
C05019=1024.414,364.393,-143.531,172.059,48.539,159.627
C05020=1024.406,364.146,-143.493,172.052,48.540,159.626
C05021=1024.398,363.900,-143.453,172.044,48.539,159.625
C05022=1024.390,363.654,-143.414,172.036,48.539,159.624
C05023=1024.382,363.406,-143.375,172.028,48.539,159.623
C05024=1024.374,363.160,-143.336,172.021,48.538,159.621
C05025=1024.365,362.913,-143.297,172.013,48.539,159.620
C05026=1024.357,362.666,-143.258,172.005,48.538,159.619
C05027=1024.349,362.419,-143.219,171.997,48.539,159.618
C05028=1024.342,362.172,-143.180,171.990,48.538,159.617
C05029=1024.334,361.926,-143.141,171.983,48.538,159.616
C05030=1024.325,361.679,-143.102,171.974,48.538,159.615
C05031=1024.317,361.432,-143.063,171.967,48.538,159.613
C05032=1024.309,361.186,-143.024,171.959,48.538,159.612
C05033=1024.302,360.939,-142.984,171.952,48.538,159.611
C05034=1024.294,360.691,-142.946,171.945,48.538,159.610
C05035=1024.285,360.444,-142.907,171.937,48.538,159.609
C05036=1024.278,360.198,-142.868,171.929,48.537,159.608
C05037=1024.269,359.951,-142.830,171.922,48.537,159.607
C05038=1024.261,359.704,-142.791,171.914,48.538,159.606
C05039=1024.254,359.457,-142.753,171.907,48.538,159.605
C05040=1024.246,359.210,-142.714,171.899,48.538,159.604
C05041=1024.237,358.963,-142.676,171.892,48.538,159.603
C05042=1024.230,358.716,-142.637,171.885,48.537,159.601
C05043=1024.222,358.469,-142.599,171.877,48.538,159.600
C05044=1024.214,358.223,-142.561,171.869,48.538,159.599
C05045=1024.206,357.975,-142.522,171.862,48.538,159.598
C05046=1024.197,357.729,-142.484,171.854,48.538,159.597
C05047=1024.190,357.482,-142.446,171.847,48.538,159.596
C05048=1024.181,357.235,-142.407,171.840,48.538,159.595
C05049=1024.174,356.988,-142.369,171.832,48.539,159.594
C05050=1024.166,356.741,-142.330,171.825,48.539,159.593
C05051=1024.158,356.495,-142.292,171.818,48.539,159.592
C05052=1024.150,356.247,-142.253,171.811,48.539,159.591
C05053=1024.143,356.000,-142.216,171.803,48.540,159.590
C05054=1024.134,355.753,-142.178,171.796,48.540,159.589
C05055=1024.126,355.507,-142.140,171.789,48.540,159.588
C05056=1024.118,355.260,-142.101,171.781,48.540,159.587
C05057=1024.111,355.012,-142.063,171.774,48.541,159.586
C05058=1024.103,354.765,-142.025,171.767,48.541,159.585
C05059=1024.095,354.519,-141.987,171.760,48.541,159.584
C05060=1024.087,354.271,-141.949,171.753,48.541,159.583
C05061=1024.079,354.025,-141.911,171.746,48.542,159.582
C05062=1024.072,353.778,-141.873,171.738,48.542,159.581
C05063=1024.063,353.531,-141.835,171.732,48.542,159.580
C05064=1024.056,353.284,-141.798,171.725,48.542,159.579
C05065=1024.048,353.036,-141.759,171.717,48.543,159.578
C05066=1024.040,352.789,-141.722,171.710,48.543,159.577
C05067=1024.032,352.542,-141.685,171.703,48.543,159.576
C05068=1024.025,352.312,-141.650,171.696,48.544,159.575
C05069=1024.018,352.082,-141.614,171.689,48.544,159.575
C05070=1024.010,351.851,-141.579,171.683,48.544,159.574
C05071=1024.003,351.621,-141.544,171.677,48.545,159.573
C05072=1023.995,351.391,-141.509,171.670,48.545,159.572
C05073=1023.989,351.160,-141.474,171.663,48.545,159.571
C05074=1023.982,350.930,-141.439,171.657,48.546,159.570
C05075=1023.974,350.700,-141.404,171.650,48.546,159.569
C05076=1023.967,350.453,-141.366,171.644,48.547,159.568
C05077=1023.959,350.206,-141.329,171.637,48.547,159.567
C05078=1023.951,349.958,-141.291,171.629,48.548,159.567
C05079=1023.944,349.711,-141.254,171.622,48.549,159.566
C05080=1023.936,349.465,-141.216,171.615,48.549,159.565
C05081=1023.929,349.218,-141.179,171.608,48.549,159.564
C05082=1023.921,348.971,-141.141,171.602,48.550,159.563
C05083=1023.913,348.724,-141.104,171.595,48.550,159.562
C05084=1023.905,348.476,-141.066,171.588,48.550,159.561
C05085=1023.898,348.229,-141.029,171.581,48.551,159.560
C05086=1023.890,347.982,-140.992,171.575,48.552,159.560
C05087=1023.883,347.734,-140.955,171.567,48.553,159.559
C05088=1023.875,347.488,-140.918,171.560,48.553,159.558
C05089=1023.868,347.240,-140.881,171.553,48.554,159.557
C05090=1023.860,346.994,-140.844,171.547,48.555,159.556
C05091=1023.852,346.747,-140.807,171.540,48.555,159.555
C05092=1023.845,346.499,-140.770,171.533,48.556,159.554
C05093=1023.837,346.252,-140.733,171.527,48.556,159.554
C05094=1023.830,346.005,-140.695,171.520,48.557,159.553
C05095=1023.822,345.758,-140.659,171.513,48.558,159.552
C05096=1023.814,345.511,-140.622,171.506,48.558,159.551
C05097=1023.807,345.264,-140.585,171.500,48.559,159.550
C05098=1023.799,345.016,-140.549,171.493,48.559,159.549
C05099=1023.792,344.769,-140.511,171.486,48.560,159.549
C05100=1023.784,344.522,-140.474,171.480,48.561,159.548
C05101=1023.776,344.275,-140.438,171.473,48.561,159.547
C05102=1023.769,344.028,-140.400,171.466,48.562,159.546
C05103=1023.762,343.780,-140.364,171.460,48.563,159.546
C05104=1023.754,343.533,-140.327,171.453,48.564,159.545
C05105=1023.747,343.286,-140.290,171.446,48.564,159.544
C05106=1023.739,343.038,-140.254,171.440,48.565,159.543
C05107=1023.731,342.791,-140.217,171.433,48.566,159.542
C05108=1023.725,342.544,-140.181,171.426,48.567,159.542
C05109=1023.717,342.297,-140.144,171.420,48.568,159.541
C05110=1023.709,342.050,-140.108,171.413,48.568,159.540
C05111=1023.702,341.802,-140.071,171.407,48.569,159.539
C05112=1023.694,341.555,-140.034,171.400,48.570,159.538
C05113=1023.687,341.309,-139.998,171.394,48.571,159.538
C05114=1023.680,341.061,-139.961,171.387,48.572,159.537
C05115=1023.672,340.813,-139.925,171.380,48.572,159.536
C05116=1023.665,340.566,-139.889,171.374,48.574,159.535
C05117=1023.657,340.320,-139.852,171.367,48.574,159.535
C05118=1023.650,340.072,-139.815,171.361,48.576,159.534
C05119=1023.643,339.825,-139.779,171.354,48.576,159.533
C05120=1023.635,339.577,-139.743,171.348,48.577,159.533
C05121=1023.628,339.331,-139.707,171.341,48.578,159.532
C05122=1023.620,339.083,-139.671,171.335,48.579,159.531
C05123=1023.613,338.836,-139.635,171.328,48.580,159.530
C05124=1023.605,338.588,-139.599,171.321,48.581,159.530
C05125=1023.598,338.341,-139.563,171.315,48.582,159.529
C05126=1023.590,338.094,-139.526,171.308,48.583,159.528
C05127=1023.583,337.846,-139.490,171.302,48.584,159.527
C05128=1023.577,337.614,-139.457,171.297,48.585,159.527
C05129=1023.569,337.382,-139.423,171.290,48.586,159.526
C05130=1023.563,337.151,-139.389,171.285,48.587,159.526
C05131=1023.555,336.919,-139.355,171.278,48.588,159.525
C05132=1023.549,336.687,-139.322,171.273,48.589,159.524
C05133=1023.541,336.455,-139.288,171.266,48.590,159.524
C05134=1023.535,336.224,-139.254,171.261,48.591,159.523
C05135=1023.528,335.992,-139.220,171.255,48.592,159.522
C05136=1023.521,335.744,-139.185,171.248,48.593,159.522
C05137=1023.513,335.497,-139.149,171.242,48.594,159.521
C05138=1023.506,335.250,-139.113,171.235,48.595,159.520
C05139=1023.499,335.002,-139.078,171.230,48.596,159.520
C05140=1023.492,334.755,-139.042,171.223,48.597,159.519
C05141=1023.484,334.508,-139.005,171.217,48.599,159.519
C05142=1023.477,334.260,-138.970,171.211,48.600,159.518
C05143=1023.470,334.013,-138.934,171.204,48.601,159.517
C05144=1023.463,333.766,-138.899,171.198,48.602,159.517
C05145=1023.455,333.518,-138.863,171.193,48.603,159.516
C05146=1023.449,333.271,-138.828,171.186,48.605,159.515
C05147=1023.441,333.023,-138.791,171.180,48.606,159.515
C05148=1023.434,332.776,-138.756,171.173,48.607,159.514
C05149=1023.427,332.529,-138.721,171.167,48.608,159.513
C05150=1023.419,332.281,-138.685,171.161,48.609,159.513
C05151=1023.412,332.034,-138.650,171.154,48.611,159.512
C05152=1023.405,331.786,-138.615,171.149,48.612,159.512
C05153=1023.398,331.539,-138.579,171.143,48.613,159.511
C05154=1023.390,331.292,-138.544,171.137,48.615,159.511
C05155=1023.383,331.044,-138.509,171.130,48.616,159.510
C05156=1023.376,330.797,-138.474,171.124,48.617,159.509
C05157=1023.368,330.549,-138.438,171.118,48.618,159.509
C05158=1023.362,330.302,-138.402,171.112,48.620,159.508
C05159=1023.354,330.055,-138.368,171.106,48.621,159.508
C05160=1023.347,329.808,-138.333,171.100,48.622,159.507
C05161=1023.340,329.560,-138.297,171.093,48.624,159.506
C05162=1023.333,329.312,-138.262,171.088,48.625,159.506
C05163=1023.326,329.065,-138.228,171.082,48.626,159.505
C05164=1023.318,328.818,-138.191,171.075,48.628,159.505
C05165=1023.311,328.570,-138.156,171.069,48.630,159.504
C05166=1023.305,328.323,-138.121,171.063,48.631,159.504
C05167=1023.297,328.076,-138.087,171.058,48.632,159.503
C05168=1023.290,327.828,-138.051,171.052,48.634,159.503
C05169=1023.283,327.580,-138.016,171.045,48.635,159.502
C05170=1023.276,327.333,-137.981,171.039,48.637,159.501
C05171=1023.269,327.086,-137.946,171.034,48.638,159.501
C05172=1023.262,326.838,-137.912,171.028,48.639,159.500
C05173=1023.255,326.591,-137.877,171.021,48.641,159.500
C05174=1023.247,326.343,-137.842,171.015,48.643,159.499
C05175=1023.240,326.096,-137.807,171.009,48.644,159.499
C05176=1023.233,325.848,-137.773,171.004,48.645,159.498
C05177=1023.226,325.601,-137.738,170.998,48.647,159.498
C05178=1023.218,325.354,-137.704,170.992,48.648,159.497
C05179=1023.211,325.105,-137.670,170.986,48.650,159.497
C05180=1023.204,324.858,-137.634,170.979,48.652,159.496
C05181=1023.196,324.611,-137.600,170.974,48.654,159.496
C05182=1023.189,324.363,-137.566,170.968,48.655,159.495
C05183=1023.182,324.116,-137.531,170.962,48.657,159.495
C05184=1023.175,323.868,-137.497,170.956,48.659,159.494
C05185=1023.168,323.621,-137.463,170.951,48.660,159.494
C05186=1023.161,323.373,-137.428,170.945,48.661,159.493
C05187=1023.154,323.126,-137.394,170.939,48.663,159.493
C05188=1023.147,322.892,-137.361,170.934,48.665,159.493
C05189=1023.139,322.658,-137.329,170.928,48.667,159.492
C05190=1023.133,322.423,-137.296,170.922,48.668,159.492
C05191=1023.126,322.189,-137.264,170.916,48.670,159.491
C05192=1023.120,321.956,-137.231,170.911,48.671,159.491
C05193=1023.113,321.721,-137.199,170.906,48.673,159.490
C05194=1023.107,321.487,-137.167,170.900,48.674,159.490
C05195=1023.099,321.253,-137.134,170.895,48.676,159.489
C05196=1023.092,321.005,-137.100,170.889,48.678,159.489
C05197=1023.086,320.757,-137.066,170.883,48.680,159.489
C05198=1023.078,320.510,-137.031,170.878,48.681,159.488
C05199=1023.071,320.262,-136.997,170.872,48.683,159.488
C05200=1023.064,320.015,-136.963,170.866,48.685,159.487
C05201=1023.058,319.768,-136.929,170.861,48.687,159.487
C05202=1023.051,319.520,-136.895,170.855,48.688,159.486
C05203=1023.043,319.273,-136.861,170.849,48.690,159.486
C05204=1023.037,319.025,-136.827,170.844,48.692,159.486
C05205=1023.030,318.777,-136.793,170.838,48.694,159.485
C05206=1023.022,318.530,-136.758,170.832,48.696,159.485
C05207=1023.016,318.282,-136.724,170.827,48.697,159.484
C05208=1023.009,318.035,-136.690,170.821,48.699,159.484
C05209=1023.002,317.787,-136.657,170.814,48.701,159.483
C05210=1022.995,317.540,-136.623,170.810,48.703,159.483
C05211=1022.988,317.292,-136.588,170.804,48.705,159.483
C05212=1022.981,317.044,-136.554,170.798,48.707,159.482
C05213=1022.974,316.797,-136.521,170.793,48.708,159.482
C05214=1022.968,316.549,-136.487,170.787,48.710,159.481
C05215=1022.961,316.302,-136.453,170.781,48.712,159.481
C05216=1022.954,316.054,-136.419,170.776,48.714,159.481
C05217=1022.947,315.807,-136.385,170.770,48.716,159.480
C05218=1022.941,315.559,-136.351,170.765,48.718,159.480
C05219=1022.933,315.311,-136.317,170.759,48.719,159.480
C05220=1022.927,315.064,-136.284,170.753,48.721,159.479
C05221=1022.920,314.816,-136.249,170.748,48.724,159.479
C05222=1022.913,314.569,-136.216,170.742,48.725,159.478
C05223=1022.906,314.322,-136.182,170.736,48.727,159.478
C05224=1022.899,314.074,-136.148,170.731,48.729,159.478
C05225=1022.893,313.826,-136.114,170.725,48.731,159.477
C05226=1022.887,313.578,-136.081,170.720,48.733,159.477
C05227=1022.879,313.331,-136.047,170.715,48.735,159.477
C05228=1022.872,313.083,-136.013,170.710,48.737,159.476
C05229=1022.866,312.836,-135.979,170.703,48.739,159.476
C05230=1022.859,312.588,-135.946,170.698,48.741,159.476
C05231=1022.853,312.340,-135.913,170.693,48.743,159.475
C05232=1022.846,312.092,-135.878,170.687,48.745,159.475
C05233=1022.840,311.845,-135.845,170.682,48.747,159.475
C05234=1022.832,311.598,-135.811,170.676,48.749,159.474
C05235=1022.826,311.350,-135.778,170.671,48.751,159.474
C05236=1022.820,311.102,-135.744,170.665,48.753,159.473
C05237=1022.813,310.855,-135.711,170.660,48.755,159.473
C05238=1022.806,310.607,-135.677,170.655,48.757,159.473
C05239=1022.800,310.360,-135.644,170.649,48.759,159.473
C05240=1022.793,310.112,-135.611,170.644,48.761,159.472
C05241=1022.786,309.865,-135.577,170.638,48.763,159.472
C05242=1022.779,309.617,-135.545,170.632,48.766,159.472
C05243=1022.772,309.370,-135.511,170.628,48.768,159.471
C05244=1022.765,309.121,-135.478,170.622,48.770,159.471
C05245=1022.758,308.874,-135.446,170.617,48.772,159.471
C05246=1022.751,308.626,-135.413,170.611,48.775,159.471
C05247=1022.744,308.379,-135.380,170.606,48.777,159.470
C05248=1022.738,308.147,-135.350,170.601,48.779,159.470
C05249=1022.731,307.916,-135.318,170.596,48.781,159.470
C05250=1022.724,307.684,-135.288,170.591,48.783,159.469
C05251=1022.718,307.452,-135.257,170.586,48.786,159.469
C05252=1022.712,307.221,-135.226,170.581,48.788,159.469
C05253=1022.705,306.989,-135.196,170.576,48.790,159.469
C05254=1022.699,306.757,-135.165,170.571,48.792,159.468
C05255=1022.692,306.526,-135.134,170.565,48.794,159.468
C05256=1022.686,306.279,-135.102,170.561,48.796,159.468
C05257=1022.679,306.030,-135.069,170.555,48.799,159.468
C05258=1022.672,305.783,-135.036,170.550,48.801,159.468
C05259=1022.665,305.536,-135.004,170.545,48.804,159.467
C05260=1022.658,305.288,-134.971,170.539,48.806,159.467
C05261=1022.652,305.040,-134.938,170.534,48.808,159.467
C05262=1022.645,304.792,-134.905,170.529,48.811,159.467
C05263=1022.638,304.544,-134.873,170.524,48.813,159.466
C05264=1022.631,304.297,-134.840,170.518,48.815,159.466
C05265=1022.624,304.048,-134.807,170.514,48.818,159.466
C05266=1022.617,303.801,-134.775,170.508,48.820,159.466
C05267=1022.611,303.554,-134.742,170.502,48.823,159.465
C05268=1022.603,303.306,-134.710,170.497,48.825,159.465
C05269=1022.597,303.058,-134.677,170.492,48.827,159.465
C05270=1022.591,302.810,-134.644,170.487,48.830,159.465
C05271=1022.584,302.563,-134.612,170.481,48.832,159.464
C05272=1022.577,302.314,-134.580,170.477,48.835,159.464
C05273=1022.571,302.067,-134.547,170.471,48.837,159.464
C05274=1022.564,301.819,-134.515,170.467,48.840,159.464
C05275=1022.558,301.572,-134.482,170.461,48.842,159.464
C05276=1022.550,301.324,-134.450,170.456,48.844,159.463
C05277=1022.544,301.076,-134.417,170.451,48.847,159.463
C05278=1022.538,300.828,-134.385,170.445,48.850,159.463
C05279=1022.531,300.581,-134.353,170.441,48.852,159.463
C05280=1022.524,300.333,-134.320,170.435,48.855,159.463
C05281=1022.517,300.085,-134.288,170.430,48.857,159.462
C05282=1022.511,299.837,-134.256,170.424,48.859,159.462
C05283=1022.505,299.589,-134.223,170.420,48.862,159.462
C05284=1022.497,299.342,-134.191,170.414,48.865,159.462
C05285=1022.492,299.094,-134.159,170.410,48.867,159.462
C05286=1022.484,298.847,-134.126,170.404,48.869,159.461
C05287=1022.478,298.598,-134.093,170.400,48.872,159.461
C05288=1022.472,298.350,-134.061,170.394,48.875,159.461
C05289=1022.465,298.103,-134.029,170.389,48.877,159.461
C05290=1022.459,297.855,-133.997,170.384,48.880,159.461
C05291=1022.452,297.607,-133.965,170.379,48.882,159.461
C05292=1022.446,297.359,-133.933,170.374,48.885,159.460
C05293=1022.439,297.111,-133.900,170.369,48.888,159.460
C05294=1022.432,296.864,-133.868,170.364,48.890,159.460
C05295=1022.426,296.616,-133.836,170.359,48.893,159.460
C05296=1022.419,296.369,-133.804,170.355,48.895,159.460
C05297=1022.413,296.120,-133.772,170.349,48.898,159.460
C05298=1022.407,295.872,-133.740,170.344,48.901,159.460
C05299=1022.400,295.625,-133.708,170.339,48.903,159.459
C05300=1022.394,295.377,-133.676,170.334,48.906,159.459
C05301=1022.387,295.129,-133.644,170.329,48.909,159.459
C05302=1022.381,294.881,-133.612,170.324,48.911,159.459
C05303=1022.375,294.634,-133.579,170.319,48.914,159.459
C05304=1022.368,294.386,-133.547,170.314,48.917,159.459
C05305=1022.362,294.138,-133.515,170.309,48.919,159.459
C05306=1022.355,293.890,-133.483,170.304,48.922,159.459
C05307=1022.349,293.642,-133.451,170.300,48.924,159.458
C05308=1022.343,293.419,-133.423,170.295,48.927,159.458
C05309=1022.337,293.197,-133.394,170.291,48.929,159.458
C05310=1022.332,292.973,-133.366,170.286,48.932,159.458
C05311=1022.326,292.751,-133.337,170.282,48.934,159.458
C05312=1022.320,292.528,-133.308,170.277,48.937,159.458
C05313=1022.314,292.305,-133.280,170.273,48.940,159.458
C05314=1022.308,292.082,-133.251,170.268,48.942,159.458
C05315=1022.303,291.860,-133.223,170.264,48.945,159.457
C05316=1022.296,291.612,-133.192,170.259,48.947,159.457
C05317=1022.289,291.364,-133.160,170.254,48.951,159.457
C05318=1022.283,291.116,-133.129,170.249,48.953,159.457
C05319=1022.276,290.868,-133.097,170.244,48.956,159.457
C05320=1022.269,290.620,-133.066,170.240,48.959,159.457
C05321=1022.262,290.372,-133.035,170.234,48.962,159.457
C05322=1022.256,290.124,-133.003,170.230,48.965,159.457
C05323=1022.250,289.876,-132.971,170.224,48.968,159.457
C05324=1022.243,289.628,-132.940,170.220,48.971,159.457
C05325=1022.236,289.380,-132.908,170.214,48.973,159.457
C05326=1022.230,289.133,-132.878,170.210,48.976,159.457
C05327=1022.224,288.885,-132.846,170.205,48.979,159.457
C05328=1022.217,288.637,-132.815,170.200,48.982,159.457
C05329=1022.210,288.389,-132.784,170.195,48.986,159.456
C05330=1022.203,288.141,-132.752,170.191,48.988,159.456
C05331=1022.198,287.893,-132.720,170.185,48.992,159.456
C05332=1022.192,287.645,-132.690,170.181,48.994,159.456
C05333=1022.185,287.397,-132.658,170.176,48.998,159.456
C05334=1022.178,287.149,-132.627,170.171,49.000,159.456
C05335=1022.172,286.901,-132.595,170.166,49.004,159.456
C05336=1022.166,286.653,-132.565,170.162,49.006,159.456
C05337=1022.159,286.405,-132.534,170.156,49.010,159.456
C05338=1022.152,286.158,-132.502,170.152,49.012,159.456
C05339=1022.146,285.909,-132.472,170.147,49.016,159.456
C05340=1022.139,285.661,-132.440,170.142,49.019,159.456
C05341=1022.133,285.414,-132.409,170.138,49.021,159.456
C05342=1022.127,285.165,-132.378,170.133,49.025,159.456
C05343=1022.120,284.918,-132.347,170.129,49.028,159.456
C05344=1022.113,284.670,-132.317,170.123,49.031,159.456
C05345=1022.107,284.422,-132.286,170.119,49.034,159.456
C05346=1022.100,284.174,-132.255,170.114,49.037,159.456
C05347=1022.093,283.926,-132.224,170.109,49.040,159.456
C05348=1022.088,283.678,-132.193,170.104,49.044,159.456
C05349=1022.081,283.430,-132.162,170.100,49.047,159.456
C05350=1022.074,283.182,-132.132,170.095,49.050,159.456
C05351=1022.067,282.934,-132.100,170.091,49.054,159.456
C05352=1022.061,282.686,-132.070,170.085,49.057,159.456
C05353=1022.055,282.437,-132.039,170.081,49.060,159.456
C05354=1022.048,282.190,-132.008,170.076,49.063,159.456
C05355=1022.041,281.942,-131.978,170.072,49.066,159.456
C05356=1022.035,281.694,-131.947,170.066,49.069,159.456
C05357=1022.028,281.446,-131.916,170.062,49.072,159.456
